LIN {X 0,Y 439.366,Z 188.757,A -85,B 0,C 180,E1 -9231.61,E2 -9231.61} C_VEL
LIN {X 0,Y 439.396,Z 188.754,A -85,B 0,C 180,E1 -9234.843,E2 -9234.843} C_VEL
LIN {X 0,Y 439.362,Z 188.757,A -85,B 0,C 180,E1 -9238.138,E2 -9238.138} C_VEL
LIN {X 0,Y 439.264,Z 188.772,A -85,B 0,C 180,E1 -9240.264,E2 -9240.264} C_VEL
LIN {X 0,Y 439.153,Z 188.786,A -85,B 0,C 180,E1 -9241.307,E2 -9241.307} C_VEL
LIN {X 0,Y 439.144,Z 192.534,A -85,B 0,C 180,E1 -9244.398,E2 -9244.398} C_VEL
LIN {X 0,Y 439.032,Z 196.208,A -85,B 0,C 180,E1 -9247.405,E2 -9247.405} C_VEL
LIN {X 0,Y 438.967,Z 200.55,A -85,B 0,C 180,E1 -9250.841,E2 -9250.841} C_VEL
LIN {X 0,Y 438.942,Z 204.965,A -85,B 0,C 180,E1 -9254.204,E2 -9254.204} C_VEL
LIN {X 0,Y 438.995,Z 210.349,A -85,B 0,C 180,E1 -9257.987,E2 -9257.987} C_VEL
LIN {X 0,Y 438.917,Z 212.924,A -85,B 0,C 180,E1 -9259.65,E2 -9259.65} C_VEL
LIN {X 0,Y 441.323,Z 223.751,A -85,B 0,C 180,E1 -9260.165,E2 -9260.165} C_VEL
LIN {X 0,Y 441.548,Z 228.336,A -85,B 0,C 180,E1 -9260.424,E2 -9260.424} C_VEL
LIN {X 0,Y 441.418,Z 237.367,A -85,B 0,C 180,E1 -9261.06,E2 -9261.06} C_VEL
LIN {X 0,Y 441.338,Z 239.701,A -85,B 0,C 180,E1 -9261.27,E2 -9261.27} C_VEL
LIN {X 0,Y 440.592,Z 243.022,A -85,B 0,C 180,E1 -9261.552,E2 -9261.552} C_VEL
LIN {X 0,Y 437.589,Z 248.036,A -85,B 0,C 180,E1 -9261.998,E2 -9261.998} C_VEL
LIN {X 0,Y 434.58,Z 252.712,A -85,B 0,C 180,E1 -9262.503,E2 -9262.503} C_VEL
LIN {X 0,Y 433.802,Z 255.354,A -85,B 0,C 180,E1 -9262.882,E2 -9262.882} C_VEL
LIN {X 0,Y 433.395,Z 261.174,A -85,B 0,C 180,E1 -9263.948,E2 -9263.948} C_VEL
LIN {X 0,Y 433.059,Z 265.059,A -85,B 0,C 180,E1 -9264.878,E2 -9264.878} C_VEL
LIN {X 0,Y 432.817,Z 269.268,A -85,B 0,C 180,E1 -9266.275,E2 -9266.275} C_VEL
LIN {X 0,Y 432.501,Z 271.224,A -85,B 0,C 180,E1 -9267.205,E2 -9267.205} C_VEL
LIN {X 0,Y 432.474,Z 272.539,A -85,B 0,C 180,E1 -9268.136,E2 -9268.136} C_VEL
LIN {X 0,Y 432.367,Z 273.322,A -85,B 0,C 180,E1 -9269.067,E2 -9269.067} C_VEL
LIN {X 0,Y 432.324,Z 273.591,A -85,B 0,C 180,E1 -9269.999,E2 -9269.999} C_VEL
LIN {X 0,Y 432.36,Z 273.368,A -85,B 0,C 180,E1 -9270.93,E2 -9270.93} C_VEL
LIN {X 0,Y 432.448,Z 272.641,A -85,B 0,C 180,E1 -9271.861,E2 -9271.861} C_VEL
LIN {X 0,Y 432.495,Z 271.382,A -85,B 0,C 180,E1 -9272.793,E2 -9272.793} C_VEL
LIN {X 0,Y 432.977,Z 268.298,A -85,B 0,C 180,E1 -9274.188,E2 -9274.188} C_VEL
LIN {X 0,Y 433.091,Z 263.642,A -85,B 0,C 180,E1 -9275.586,E2 -9275.586} C_VEL
LIN {X 0,Y 433.453,Z 260.509,A -85,B 0,C 180,E1 -9276.282,E2 -9276.282} C_VEL
LIN {X 0,Y 433.76,Z 253.871,A -85,B 0,C 180,E1 -9277.446,E2 -9277.446} C_VEL
LIN {X 0,Y 434.169,Z 246.685,A -85,B 0,C 180,E1 -9278.376,E2 -9278.376} C_VEL
LIN {X 0,Y 434.424,Z 239.235,A -85,B 0,C 180,E1 -9279.124,E2 -9279.124} C_VEL
LIN {X 0,Y 434.667,Z 230.594,A -85,B 0,C 180,E1 -9279.773,E2 -9279.773} C_VEL
LIN {X 0,Y 434.533,Z 225.553,A -85,B 0,C 180,E1 -9280.07,E2 -9280.07} C_VEL
LIN {X 0,Y 432.434,Z 216.056,A -85,B 0,C 180,E1 -9280.549,E2 -9280.549} C_VEL
LIN {X 0,Y 431.91,Z 213.531,A -85,B 0,C 180,E1 -9280.665,E2 -9280.665} C_VEL
LIN {X 0,Y 431.872,Z 209.743,A -85,B 0,C 180,E1 -9283.168,E2 -9283.168} C_VEL
LIN {X 0,Y 431.93,Z 205.419,A -85,B 0,C 180,E1 -9286.26,E2 -9286.26} C_VEL
LIN {X 0,Y 431.936,Z 201.432,A -85,B 0,C 180,E1 -9289.314,E2 -9289.314} C_VEL
LIN {X 0,Y 432.007,Z 198.074,A -85,B 0,C 180,E1 -9291.983,E2 -9291.983} C_VEL
LIN {X 0,Y 432.063,Z 194.327,A -85,B 0,C 180,E1 -9295.017,E2 -9295.017} C_VEL
LIN {X 0,Y 432.113,Z 191.814,A -85,B 0,C 180,E1 -9297.089,E2 -9297.089} C_VEL
LIN {X 0,Y 432.131,Z 190.006,A -85,B 0,C 180,E1 -9298.569,E2 -9298.569} C_VEL
LIN {X 0,Y 432.145,Z 189.659,A -85,B 0,C 180,E1 -9299.2,E2 -9299.2} C_VEL
LIN {X 0,Y 432.301,Z 189.637,A -85,B 0,C 180,E1 -9301.346,E2 -9301.346} C_VEL
LIN {X 0,Y 432.336,Z 189.63,A -85,B 0,C 180,E1 -9304.676,E2 -9304.676} C_VEL
LIN {X 0,Y 432.341,Z 189.629,A -85,B 0,C 180,E1 -9308.148,E2 -9308.148} C_VEL
LIN {X 0,Y 432.328,Z 189.632,A -85,B 0,C 180,E1 -9311.601,E2 -9311.601} C_VEL
LIN {X 0,Y 432.334,Z 189.628,A -85,B 0,C 180,E1 -9314.345,E2 -9314.345} C_VEL
LIN {X 0,Y 432.313,Z 189.635,A -85,B 0,C 180,E1 -9317.014,E2 -9317.014} C_VEL
LIN {X 0,Y 432.336,Z 189.627,A -85,B 0,C 180,E1 -9319.818,E2 -9319.818} C_VEL
LIN {X 0,Y 432.308,Z 189.634,A -85,B 0,C 180,E1 -9323.022,E2 -9323.022} C_VEL
LIN {X 0,Y 432.351,Z 189.627,A -85,B 0,C 180,E1 -9325.995,E2 -9325.995} C_VEL
LIN {X 0,Y 432.386,Z 189.622,A -85,B 0,C 180,E1 -9329.743,E2 -9329.743} C_VEL
LIN {X 0,Y 432.39,Z 189.622,A -85,B 0,C 180,E1 -9333.371,E2 -9333.371} C_VEL
LIN {X 0,Y 432.361,Z 189.626,A -85,B 0,C 180,E1 -9336.023,E2 -9336.023} C_VEL
LIN {X 0,Y 432.34,Z 189.625,A -85,B 0,C 180,E1 -9339.045,E2 -9339.045} C_VEL
LIN {X 0,Y 432.368,Z 189.629,A -85,B 0,C 180,E1 -9342.011,E2 -9342.011} C_VEL
LIN {X 0,Y 432.391,Z 189.615,A -85,B 0,C 180,E1 -9344.926,E2 -9344.926} C_VEL
LIN {X 0,Y 432.448,Z 189.617,A -85,B 0,C 180,E1 -9347.803,E2 -9347.803} C_VEL
LIN {X 0,Y 432.481,Z 189.614,A -85,B 0,C 180,E1 -9351.59,E2 -9351.59} C_VEL
LIN {X 0,Y 432.582,Z 189.594,A -85,B 0,C 180,E1 -9354.406,E2 -9354.406} C_VEL
LIN {X 0,Y 432.595,Z 189.595,A -85,B 0,C 180,E1 -9358.138,E2 -9358.138} C_VEL
LIN {X 0,Y 432.72,Z 189.573,A -85,B 0,C 180,E1 -9360,E2 -9360} C_VEL
LIN {X 0,Y 432.578,Z 189.604,A -85,B 0,C 180,E1 -9362.794,E2 -9362.794} C_VEL
LIN {X 0,Y 432.556,Z 189.604,A -85,B 0,C 180,E1 -9366.531,E2 -9366.531} C_VEL
LIN {X 0,Y 432.429,Z 189.613,A -85,B 0,C 180,E1 -9369.353,E2 -9369.353} C_VEL
LIN {X 0,Y 432.419,Z 189.616,A -85,B 0,C 180,E1 -9372.804,E2 -9372.804} C_VEL
LIN {X 0,Y 432.399,Z 189.622,A -85,B 0,C 180,E1 -9376.479,E2 -9376.479} C_VEL
LIN {X 0,Y 432.327,Z 189.637,A -85,B 0,C 180,E1 -9379.961,E2 -9379.961} C_VEL
LIN {X 0,Y 432.299,Z 189.634,A -85,B 0,C 180,E1 -9382.965,E2 -9382.965} C_VEL
LIN {X 0,Y 432.306,Z 189.638,A -85,B 0,C 180,E1 -9386.036,E2 -9386.036} C_VEL
LIN {X 0,Y 432.312,Z 189.635,A -85,B 0,C 180,E1 -9389.19,E2 -9389.19} C_VEL
LIN {X 0,Y 432.312,Z 189.632,A -85,B 0,C 180,E1 -9392.444,E2 -9392.444} C_VEL
LIN {X 0,Y 432.332,Z 189.634,A -85,B 0,C 180,E1 -9395.632,E2 -9395.632} C_VEL
LIN {X 0,Y 432.32,Z 189.636,A -85,B 0,C 180,E1 -9398.714,E2 -9398.714} C_VEL
LIN {X 0,Y 432.311,Z 189.634,A -85,B 0,C 180,E1 -9401.8,E2 -9401.8} C_VEL
LIN {X 0,Y 432.326,Z 189.632,A -85,B 0,C 180,E1 -9404.349,E2 -9404.349} C_VEL
LIN {X 0,Y 432.313,Z 189.631,A -85,B 0,C 180,E1 -9407.017,E2 -9407.017} C_VEL
LIN {X 0,Y 432.327,Z 189.634,A -85,B 0,C 180,E1 -9409.822,E2 -9409.822} C_VEL
LIN {X 0,Y 432.318,Z 189.693,A -85,B 0,C 180,E1 -9413.098,E2 -9413.098} C_VEL
LIN {X 0,Y 434.697,Z 199.485,A -85,B 0,C 180,E1 -9415.753,E2 -9415.753} C_VEL
LIN {X 0,Y 437.238,Z 210.934,A -85,B 0,C 180,E1 -9418.615,E2 -9418.615} C_VEL
LIN {X 0,Y 437.708,Z 214.124,A -85,B 0,C 180,E1 -9419.352,E2 -9419.352} C_VEL
LIN {X 0,Y 436.282,Z 228.623,A -85,B 0,C 180,E1 -9422.374,E2 -9422.374} C_VEL
LIN {X 0,Y 434.667,Z 247.312,A -85,B 0,C 180,E1 -9426.159,E2 -9426.159} C_VEL
LIN {X 0,Y 433.52,Z 264.525,A -85,B 0,C 180,E1 -9429.603,E2 -9429.603} C_VEL
LIN {X 0,Y 432.462,Z 282.864,A -85,B 0,C 180,E1 -9433.355,E2 -9433.355} C_VEL
LIN {X 0,Y 432.406,Z 284.264,A -85,B 0,C 180,E1 -9433.649,E2 -9433.649} C_VEL
LIN {X 0,Y 434.151,Z 302.397,A -85,B 0,C 180,E1 -9434.163,E2 -9434.163} C_VEL
LIN {X 0,Y 434.663,Z 314.357,A -85,B 0,C 180,E1 -9434.648,E2 -9434.648} C_VEL
LIN {X 0,Y 434.181,Z 327.38,A -85,B 0,C 180,E1 -9435.351,E2 -9435.351} C_VEL
LIN {X 0,Y 433.629,Z 339.016,A -85,B 0,C 180,E1 -9436.171,E2 -9436.171} C_VEL
LIN {X 0,Y 433.07,Z 349.53,A -85,B 0,C 180,E1 -9437.108,E2 -9437.108} C_VEL
LIN {X 0,Y 432.534,Z 360.155,A -85,B 0,C 180,E1 -9438.283,E2 -9438.283} C_VEL
LIN {X 0,Y 432.099,Z 368.825,A -85,B 0,C 180,E1 -9439.458,E2 -9439.458} C_VEL
LIN {X 0,Y 431.747,Z 377.221,A -85,B 0,C 180,E1 -9440.869,E2 -9440.869} C_VEL
LIN {X 0,Y 431.526,Z 383.96,A -85,B 0,C 180,E1 -9442.28,E2 -9442.28} C_VEL
LIN {X 0,Y 431.39,Z 389.034,A -85,B 0,C 180,E1 -9443.609,E2 -9443.609} C_VEL
LIN {X 0,Y 431.437,Z 392.806,A -85,B 0,C 180,E1 -9444.861,E2 -9444.861} C_VEL
LIN {X 0,Y 431.391,Z 395.987,A -85,B 0,C 180,E1 -9446.265,E2 -9446.265} C_VEL
LIN {X 0,Y 431.423,Z 397.549,A -85,B 0,C 180,E1 -9447.2,E2 -9447.2} C_VEL
LIN {X 0,Y 431.413,Z 398.638,A -85,B 0,C 180,E1 -9448.134,E2 -9448.134} C_VEL
LIN {X 0,Y 431.419,Z 399.29,A -85,B 0,C 180,E1 -9449.068,E2 -9449.068} C_VEL
LIN {X 0,Y 431.413,Z 399.531,A -85,B 0,C 180,E1 -9450.001,E2 -9450.001} C_VEL
LIN {X 0,Y 431.42,Z 399.348,A -85,B 0,C 180,E1 -9450.935,E2 -9450.935} C_VEL
LIN {X 0,Y 431.405,Z 398.699,A -85,B 0,C 180,E1 -9451.868,E2 -9451.868} C_VEL
LIN {X 0,Y 431.429,Z 397.639,A -85,B 0,C 180,E1 -9452.802,E2 -9452.802} C_VEL
LIN {X 0,Y 431.397,Z 396.16,A -85,B 0,C 180,E1 -9453.737,E2 -9453.737} C_VEL
LIN {X 0,Y 431.445,Z 393.062,A -85,B 0,C 180,E1 -9455.141,E2 -9455.141} C_VEL
LIN {X 0,Y 431.44,Z 388.87,A -85,B 0,C 180,E1 -9456.549,E2 -9456.549} C_VEL
LIN {X 0,Y 431.603,Z 382.413,A -85,B 0,C 180,E1 -9458.193,E2 -9458.193} C_VEL
LIN {X 0,Y 431.894,Z 375.417,A -85,B 0,C 180,E1 -9459.603,E2 -9459.603} C_VEL
LIN {X 0,Y 432.299,Z 366.74,A -85,B 0,C 180,E1 -9461.014,E2 -9461.014} C_VEL
LIN {X 0,Y 432.934,Z 355.922,A -85,B 0,C 180,E1 -9462.422,E2 -9462.422} C_VEL
LIN {X 0,Y 433.518,Z 345.135,A -85,B 0,C 180,E1 -9463.549,E2 -9463.549} C_VEL
LIN {X 0,Y 434.312,Z 333.445,A -85,B 0,C 180,E1 -9464.527,E2 -9464.527} C_VEL
LIN {X 0,Y 435.048,Z 321.115,A -85,B 0,C 180,E1 -9465.34,E2 -9465.34} C_VEL
LIN {X 0,Y 435.317,Z 311.088,A -85,B 0,C 180,E1 -9465.871,E2 -9465.871} C_VEL
LIN {X 0,Y 434.635,Z 297.333,A -85,B 0,C 180,E1 -9466.457,E2 -9466.457} C_VEL
LIN {X 0,Y 432.565,Z 280.937,A -85,B 0,C 180,E1 -9467.036,E2 -9467.036} C_VEL
LIN {X 0,Y 433.575,Z 263.253,A -85,B 0,C 180,E1 -9470.645,E2 -9470.645} C_VEL
LIN {X 0,Y 434.783,Z 246.074,A -85,B 0,C 180,E1 -9474.09,E2 -9474.09} C_VEL
LIN {X 0,Y 436.367,Z 227.495,A -85,B 0,C 180,E1 -9477.845,E2 -9477.845} C_VEL
LIN {X 0,Y 437.662,Z 214.036,A -85,B 0,C 180,E1 -9480.654,E2 -9480.654} C_VEL
LIN {X 0,Y 436.57,Z 207.954,A -85,B 0,C 180,E1 -9482.09,E2 -9482.09} C_VEL
LIN {X 0,Y 433.916,Z 196.164,A -85,B 0,C 180,E1 -9485.099,E2 -9485.099} C_VEL
LIN {X 0,Y 432.312,Z 189.638,A -85,B 0,C 180,E1 -9486.942,E2 -9486.942} C_VEL
LIN {X 0,Y 432.338,Z 189.632,A -85,B 0,C 180,E1 -9490.18,E2 -9490.18} C_VEL
LIN {X 0,Y 432.322,Z 189.634,A -85,B 0,C 180,E1 -9493.061,E2 -9493.061} C_VEL
LIN {X 0,Y 432.338,Z 189.634,A -85,B 0,C 180,E1 -9495.665,E2 -9495.665} C_VEL
LIN {X 0,Y 432.338,Z 189.633,A -85,B 0,C 180,E1 -9498.398,E2 -9498.398} C_VEL
LIN {X 0,Y 432.341,Z 189.757,A -85,B 0,C 180,E1 -9500.924,E2 -9500.924} C_VEL
LIN {X 0,Y 433.904,Z 196.549,A -85,B 0,C 180,E1 -9503.694,E2 -9503.694} C_VEL
LIN {X 0,Y 434.42,Z 199.762,A -85,B 0,C 180,E1 -9504.948,E2 -9504.948} C_VEL
LIN {X 0,Y 434.339,Z 204.343,A -85,B 0,C 180,E1 -9506.623,E2 -9506.623} C_VEL
LIN {X 0,Y 433.832,Z 213.134,A -85,B 0,C 180,E1 -9509.855,E2 -9509.855} C_VEL
LIN {X 0,Y 433.682,Z 220.548,A -85,B 0,C 180,E1 -9512.493,E2 -9512.493} C_VEL
LIN {X 0,Y 433.348,Z 229.943,A -85,B 0,C 180,E1 -9516.081,E2 -9516.081} C_VEL
LIN {X 0,Y 433.048,Z 239.208,A -85,B 0,C 180,E1 -9519.578,E2 -9519.578} C_VEL
LIN {X 0,Y 432.859,Z 246.938,A -85,B 0,C 180,E1 -9522.52,E2 -9522.52} C_VEL
LIN {X 0,Y 432.823,Z 248.27,A -85,B 0,C 180,E1 -9523.028,E2 -9523.028} C_VEL
LIN {X 0,Y 436.157,Z 261.185,A -85,B 0,C 180,E1 -9523.67,E2 -9523.67} C_VEL
LIN {X 0,Y 436.8,Z 264.746,A -85,B 0,C 180,E1 -9523.862,E2 -9523.862} C_VEL
LIN {X 0,Y 436.163,Z 278.327,A -85,B 0,C 180,E1 -9524.581,E2 -9524.581} C_VEL
LIN {X 0,Y 435.563,Z 289.849,A -85,B 0,C 180,E1 -9525.379,E2 -9525.379} C_VEL
LIN {X 0,Y 434.867,Z 300.72,A -85,B 0,C 180,E1 -9526.328,E2 -9526.328} C_VEL
LIN {X 0,Y 434.171,Z 310.523,A -85,B 0,C 180,E1 -9527.377,E2 -9527.377} C_VEL
LIN {X 0,Y 433.522,Z 319.523,A -85,B 0,C 180,E1 -9528.546,E2 -9528.546} C_VEL
LIN {X 0,Y 433.014,Z 326.938,A -85,B 0,C 180,E1 -9529.716,E2 -9529.716} C_VEL
LIN {X 0,Y 432.504,Z 334.208,A -85,B 0,C 180,E1 -9531.12,E2 -9531.12} C_VEL
LIN {X 0,Y 432.099,Z 340.07,A -85,B 0,C 180,E1 -9532.524,E2 -9532.524} C_VEL
LIN {X 0,Y 431.763,Z 344.689,A -85,B 0,C 180,E1 -9533.927,E2 -9533.927} C_VEL
LIN {X 0,Y 431.703,Z 348.178,A -85,B 0,C 180,E1 -9535.331,E2 -9535.331} C_VEL
LIN {X 0,Y 431.565,Z 349.968,A -85,B 0,C 180,E1 -9536.265,E2 -9536.265} C_VEL
LIN {X 0,Y 431.472,Z 351.286,A -85,B 0,C 180,E1 -9537.199,E2 -9537.199} C_VEL
LIN {X 0,Y 431.4,Z 352.199,A -85,B 0,C 180,E1 -9538.133,E2 -9538.133} C_VEL
LIN {X 0,Y 431.318,Z 352.722,A -85,B 0,C 180,E1 -9539.066,E2 -9539.066} C_VEL
LIN {X 0,Y 431.289,Z 352.813,A -85,B 0,C 180,E1 -9540,E2 -9540} C_VEL
LIN {X 0,Y 431.314,Z 351.753,A -85,B 0,C 180,E1 -9541.868,E2 -9541.868} C_VEL
LIN {X 0,Y 431.417,Z 350.62,A -85,B 0,C 180,E1 -9542.801,E2 -9542.801} C_VEL
LIN {X 0,Y 431.478,Z 348.099,A -85,B 0,C 180,E1 -9544.203,E2 -9544.203} C_VEL
LIN {X 0,Y 431.584,Z 344.559,A -85,B 0,C 180,E1 -9545.607,E2 -9545.607} C_VEL
LIN {X 0,Y 431.809,Z 339.391,A -85,B 0,C 180,E1 -9547.141,E2 -9547.141} C_VEL
LIN {X 0,Y 432.139,Z 332.851,A -85,B 0,C 180,E1 -9548.652,E2 -9548.652} C_VEL
LIN {X 0,Y 432.552,Z 325.23,A -85,B 0,C 180,E1 -9550.059,E2 -9550.059} C_VEL
LIN {X 0,Y 433.107,Z 315.679,A -85,B 0,C 180,E1 -9551.466,E2 -9551.466} C_VEL
LIN {X 0,Y 433.669,Z 305.897,A -85,B 0,C 180,E1 -9552.637,E2 -9552.637} C_VEL
LIN {X 0,Y 434.238,Z 294.872,A -85,B 0,C 180,E1 -9553.701,E2 -9553.701} C_VEL
LIN {X 0,Y 434.789,Z 282.839,A -85,B 0,C 180,E1 -9554.629,E2 -9554.629} C_VEL
LIN {X 0,Y 435.382,Z 269.906,A -85,B 0,C 180,E1 -9555.387,E2 -9555.387} C_VEL
LIN {X 0,Y 435.38,Z 262.377,A -85,B 0,C 180,E1 -9555.747,E2 -9555.747} C_VEL
LIN {X 0,Y 432.829,Z 248.974,A -85,B 0,C 180,E1 -9556.301,E2 -9556.301} C_VEL
LIN {X 0,Y 432.198,Z 245.514,A -85,B 0,C 180,E1 -9556.427,E2 -9556.427} C_VEL
LIN {X 0,Y 432.364,Z 236.205,A -85,B 0,C 180,E1 -9559.959,E2 -9559.959} C_VEL
LIN {X 0,Y 432.545,Z 228.361,A -85,B 0,C 180,E1 -9562.952,E2 -9562.952} C_VEL
LIN {X 0,Y 432.692,Z 220.375,A -85,B 0,C 180,E1 -9566.011,E2 -9566.011} C_VEL
LIN {X 0,Y 432.957,Z 212.189,A -85,B 0,C 180,E1 -9569.142,E2 -9569.142} C_VEL
LIN {X 0,Y 433.133,Z 203.812,A -85,B 0,C 180,E1 -9572.375,E2 -9572.375} C_VEL
LIN {X 0,Y 433.269,Z 196.593,A -85,B 0,C 180,E1 -9575.159,E2 -9575.159} C_VEL
LIN {X 0,Y 432.669,Z 191.204,A -85,B 0,C 180,E1 -9577.256,E2 -9577.256} C_VEL
LIN {X 0,Y 432.379,Z 189.628,A -85,B 0,C 180,E1 -9577.906,E2 -9577.906} C_VEL
LIN {X 0,Y 432.326,Z 189.633,A -85,B 0,C 180,E1 -9580.561,E2 -9580.561} C_VEL
LIN {X 0,Y 432.319,Z 189.634,A -85,B 0,C 180,E1 -9583.061,E2 -9583.061} C_VEL
LIN {X 0,Y 432.338,Z 189.631,A -85,B 0,C 180,E1 -9585.664,E2 -9585.664} C_VEL
LIN {X 0,Y 432.338,Z 189.631,A -85,B 0,C 180,E1 -9588.398,E2 -9588.398} C_VEL
LIN {X 0,Y 432.33,Z 189.634,A -85,B 0,C 180,E1 -9591.848,E2 -9591.848} C_VEL
LIN {X 0,Y 432.33,Z 189.636,A -85,B 0,C 180,E1 -9595.321,E2 -9595.321} C_VEL
LIN {X 0,Y 432.3,Z 189.639,A -85,B 0,C 180,E1 -9598.651,E2 -9598.651} C_VEL
LIN {X 0,Y 432.125,Z 189.881,A -85,B 0,C 180,E1 -9601.432,E2 -9601.432} C_VEL
LIN {X 0,Y 432.115,Z 192.93,A -85,B 0,C 180,E1 -9603.95,E2 -9603.95} C_VEL
LIN {X 0,Y 432.005,Z 196.684,A -85,B 0,C 180,E1 -9607.017,E2 -9607.017} C_VEL
LIN {X 0,Y 431.941,Z 201.27,A -85,B 0,C 180,E1 -9610.684,E2 -9610.684} C_VEL
LIN {X 0,Y 431.898,Z 205.538,A -85,B 0,C 180,E1 -9613.94,E2 -9613.94} C_VEL
LIN {X 0,Y 431.944,Z 211,A -85,B 0,C 180,E1 -9617.788,E2 -9617.788} C_VEL
LIN {X 0,Y 431.898,Z 213.618,A -85,B 0,C 180,E1 -9619.451,E2 -9619.451} C_VEL
LIN {X 0,Y 434.257,Z 224.071,A -85,B 0,C 180,E1 -9619.939,E2 -9619.939} C_VEL
LIN {X 0,Y 434.685,Z 227.626,A -85,B 0,C 180,E1 -9620.143,E2 -9620.143} C_VEL
LIN {X 0,Y 434.506,Z 236.893,A -85,B 0,C 180,E1 -9620.774,E2 -9620.774} C_VEL
LIN {X 0,Y 434.227,Z 244.517,A -85,B 0,C 180,E1 -9621.472,E2 -9621.472} C_VEL
LIN {X 0,Y 433.86,Z 251.526,A -85,B 0,C 180,E1 -9622.319,E2 -9622.319} C_VEL
LIN {X 0,Y 433.802,Z 255.354,A -85,B 0,C 180,E1 -9622.882,E2 -9622.882} C_VEL
LIN {X 0,Y 433.001,Z 257.885,A -85,B 0,C 180,E1 -9623.282,E2 -9623.282} C_VEL
LIN {X 0,Y 429.88,Z 261.704,A -85,B 0,C 180,E1 -9623.901,E2 -9623.901} C_VEL
LIN {X 0,Y 426.797,Z 265.096,A -85,B 0,C 180,E1 -9624.567,E2 -9624.567} C_VEL
LIN {X 0,Y 426.058,Z 266.865,A -85,B 0,C 180,E1 -9625.034,E2 -9625.034} C_VEL
LIN {X 0,Y 425.815,Z 270.255,A -85,B 0,C 180,E1 -9626.213,E2 -9626.213} C_VEL
LIN {X 0,Y 425.487,Z 272.204,A -85,B 0,C 180,E1 -9627.158,E2 -9627.158} C_VEL
LIN {X 0,Y 425.456,Z 273.515,A -85,B 0,C 180,E1 -9628.106,E2 -9628.106} C_VEL
LIN {X 0,Y 425.345,Z 274.296,A -85,B 0,C 180,E1 -9629.052,E2 -9629.052} C_VEL
LIN {X 0,Y 425.3,Z 274.565,A -85,B 0,C 180,E1 -9629.999,E2 -9629.999} C_VEL
LIN {X 0,Y 425.339,Z 274.342,A -85,B 0,C 180,E1 -9630.946,E2 -9630.946} C_VEL
LIN {X 0,Y 425.432,Z 273.616,A -85,B 0,C 180,E1 -9631.892,E2 -9631.892} C_VEL
LIN {X 0,Y 425.482,Z 272.362,A -85,B 0,C 180,E1 -9632.839,E2 -9632.839} C_VEL
LIN {X 0,Y 425.981,Z 269.288,A -85,B 0,C 180,E1 -9634.256,E2 -9634.256} C_VEL
LIN {X 0,Y 426.098,Z 264.654,A -85,B 0,C 180,E1 -9635.678,E2 -9635.678} C_VEL
LIN {X 0,Y 426.473,Z 261.542,A -85,B 0,C 180,E1 -9636.385,E2 -9636.385} C_VEL
LIN {X 0,Y 426.807,Z 254.956,A -85,B 0,C 180,E1 -9637.568,E2 -9637.568} C_VEL
LIN {X 0,Y 427.234,Z 247.821,A -85,B 0,C 180,E1 -9638.513,E2 -9638.513} C_VEL
LIN {X 0,Y 427.507,Z 240.315,A -85,B 0,C 180,E1 -9639.284,E2 -9639.284} C_VEL
LIN {X 0,Y 427.786,Z 231.984,A -85,B 0,C 180,E1 -9639.932,E2 -9639.932} C_VEL
LIN {X 0,Y 427.696,Z 227.044,A -85,B 0,C 180,E1 -9640.233,E2 -9640.233} C_VEL
LIN {X 0,Y 425.517,Z 216.936,A -85,B 0,C 180,E1 -9640.76,E2 -9640.76} C_VEL
LIN {X 0,Y 424.854,Z 214.126,A -85,B 0,C 180,E1 -9640.905,E2 -9640.905} C_VEL
LIN {X 0,Y 424.827,Z 210.378,A -85,B 0,C 180,E1 -9643.39,E2 -9643.39} C_VEL
LIN {X 0,Y 424.894,Z 206.183,A -85,B 0,C 180,E1 -9646.391,E2 -9646.391} C_VEL
LIN {X 0,Y 424.887,Z 202.17,A -85,B 0,C 180,E1 -9649.467,E2 -9649.467} C_VEL
LIN {X 0,Y 424.95,Z 198.543,A -85,B 0,C 180,E1 -9652.356,E2 -9652.356} C_VEL
LIN {X 0,Y 425.048,Z 194.746,A -85,B 0,C 180,E1 -9655.46,E2 -9655.46} C_VEL
LIN {X 0,Y 425.101,Z 190.885,A -85,B 0,C 180,E1 -9658.647,E2 -9658.647} C_VEL
LIN {X 0,Y 425.239,Z 190.515,A -85,B 0,C 180,E1 -9660.818,E2 -9660.818} C_VEL
LIN {X 0,Y 425.308,Z 190.506,A -85,B 0,C 180,E1 -9664.287,E2 -9664.287} C_VEL
LIN {X 0,Y 425.281,Z 190.511,A -85,B 0,C 180,E1 -9667.692,E2 -9667.692} C_VEL
LIN {X 0,Y 425.276,Z 190.509,A -85,B 0,C 180,E1 -9670.519,E2 -9670.519} C_VEL
LIN {X 0,Y 425.257,Z 190.513,A -85,B 0,C 180,E1 -9673.35,E2 -9673.35} C_VEL
LIN {X 0,Y 425.25,Z 190.513,A -85,B 0,C 180,E1 -9676.648,E2 -9676.648} C_VEL
LIN {X 0,Y 425.289,Z 190.505,A -85,B 0,C 180,E1 -9679.873,E2 -9679.873} C_VEL
LIN {X 0,Y 425.277,Z 190.51,A -85,B 0,C 180,E1 -9682.486,E2 -9682.486} C_VEL
LIN {X 0,Y 425.299,Z 190.504,A -85,B 0,C 180,E1 -9685.816,E2 -9685.816} C_VEL
LIN {X 0,Y 425.295,Z 190.505,A -85,B 0,C 180,E1 -9689.235,E2 -9689.235} C_VEL
LIN {X 0,Y 425.341,Z 190.504,A -85,B 0,C 180,E1 -9692.442,E2 -9692.442} C_VEL
LIN {X 0,Y 425.341,Z 190.496,A -85,B 0,C 180,E1 -9695.601,E2 -9695.601} C_VEL
LIN {X 0,Y 425.283,Z 190.504,A -85,B 0,C 180,E1 -9698.681,E2 -9698.681} C_VEL
LIN {X 0,Y 425.323,Z 190.506,A -85,B 0,C 180,E1 -9701.702,E2 -9701.702} C_VEL
LIN {X 0,Y 425.345,Z 190.492,A -85,B 0,C 180,E1 -9704.67,E2 -9704.67} C_VEL
LIN {X 0,Y 425.401,Z 190.497,A -85,B 0,C 180,E1 -9707.598,E2 -9707.598} C_VEL
LIN {X 0,Y 425.431,Z 190.491,A -85,B 0,C 180,E1 -9711.45,E2 -9711.45} C_VEL
LIN {X 0,Y 425.538,Z 190.471,A -85,B 0,C 180,E1 -9714.313,E2 -9714.313} C_VEL
LIN {X 0,Y 425.564,Z 190.471,A -85,B 0,C 180,E1 -9718.107,E2 -9718.107} C_VEL
LIN {X 0,Y 425.69,Z 190.449,A -85,B 0,C 180,E1 -9720,E2 -9720} C_VEL
LIN {X 0,Y 425.531,Z 190.481,A -85,B 0,C 180,E1 -9722.84,E2 -9722.84} C_VEL
LIN {X 0,Y 425.515,Z 190.483,A -85,B 0,C 180,E1 -9726.639,E2 -9726.639} C_VEL
LIN {X 0,Y 425.387,Z 190.489,A -85,B 0,C 180,E1 -9729.51,E2 -9729.51} C_VEL
LIN {X 0,Y 425.381,Z 190.492,A -85,B 0,C 180,E1 -9732.904,E2 -9732.904} C_VEL
LIN {X 0,Y 425.349,Z 190.499,A -85,B 0,C 180,E1 -9736.605,E2 -9736.605} C_VEL
LIN {X 0,Y 425.316,Z 190.506,A -85,B 0,C 180,E1 -9739.636,E2 -9739.636} C_VEL
LIN {X 0,Y 425.275,Z 190.512,A -85,B 0,C 180,E1 -9742.339,E2 -9742.339} C_VEL
LIN {X 0,Y 425.248,Z 190.516,A -85,B 0,C 180,E1 -9745.448,E2 -9745.448} C_VEL
LIN {X 0,Y 425.289,Z 190.508,A -85,B 0,C 180,E1 -9748.859,E2 -9748.859} C_VEL
LIN {X 0,Y 425.254,Z 190.513,A -85,B 0,C 180,E1 -9751.928,E2 -9751.928} C_VEL
LIN {X 0,Y 425.287,Z 190.51,A -85,B 0,C 180,E1 -9755.337,E2 -9755.337} C_VEL
LIN {X 0,Y 425.274,Z 190.516,A -85,B 0,C 180,E1 -9758.901,E2 -9758.901} C_VEL
LIN {X 0,Y 425.271,Z 190.511,A -85,B 0,C 180,E1 -9761.958,E2 -9761.958} C_VEL
LIN {X 0,Y 425.277,Z 190.51,A -85,B 0,C 180,E1 -9765.284,E2 -9765.284} C_VEL
LIN {X 0,Y 425.267,Z 190.507,A -85,B 0,C 180,E1 -9768.623,E2 -9768.623} C_VEL
LIN {X 0,Y 425.3,Z 190.503,A -85,B 0,C 180,E1 -9771.104,E2 -9771.104} C_VEL
LIN {X 0,Y 425.309,Z 190.713,A -85,B 0,C 180,E1 -9772.684,E2 -9772.684} C_VEL
LIN {X 0,Y 427.903,Z 201.469,A -85,B 0,C 180,E1 -9775.679,E2 -9775.679} C_VEL
LIN {X 0,Y 430.377,Z 212.6,A -85,B 0,C 180,E1 -9778.498,E2 -9778.498} C_VEL
LIN {X 0,Y 430.803,Z 216.222,A -85,B 0,C 180,E1 -9779.351,E2 -9779.351} C_VEL
LIN {X 0,Y 429.104,Z 232.027,A -85,B 0,C 180,E1 -9782.705,E2 -9782.705} C_VEL
LIN {X 0,Y 427.623,Z 249.211,A -85,B 0,C 180,E1 -9786.257,E2 -9786.257} C_VEL
LIN {X 0,Y 426.408,Z 266.239,A -85,B 0,C 180,E1 -9789.751,E2 -9789.751} C_VEL
LIN {X 0,Y 425.359,Z 283.693,A -85,B 0,C 180,E1 -9793.418,E2 -9793.418} C_VEL
LIN {X 0,Y 427.186,Z 302.416,A -85,B 0,C 180,E1 -9793.96,E2 -9793.96} C_VEL
LIN {X 0,Y 427.699,Z 315.433,A -85,B 0,C 180,E1 -9794.514,E2 -9794.514} C_VEL
LIN {X 0,Y 427.147,Z 328.088,A -85,B 0,C 180,E1 -9795.226,E2 -9795.226} C_VEL
LIN {X 0,Y 426.604,Z 339.456,A -85,B 0,C 180,E1 -9796.06,E2 -9796.06} C_VEL
LIN {X 0,Y 426.03,Z 349.777,A -85,B 0,C 180,E1 -9797.01,E2 -9797.01} C_VEL
LIN {X 0,Y 425.505,Z 359.342,A -85,B 0,C 180,E1 -9798.086,E2 -9798.086} C_VEL
LIN {X 0,Y 425.05,Z 368.084,A -85,B 0,C 180,E1 -9799.281,E2 -9799.281} C_VEL
LIN {X 0,Y 424.693,Z 376.568,A -85,B 0,C 180,E1 -9800.716,E2 -9800.716} C_VEL
LIN {X 0,Y 424.438,Z 383.356,A -85,B 0,C 180,E1 -9802.15,E2 -9802.15} C_VEL
LIN {X 0,Y 424.292,Z 388.951,A -85,B 0,C 180,E1 -9803.641,E2 -9803.641} C_VEL
LIN {X 0,Y 424.32,Z 393.495,A -85,B 0,C 180,E1 -9805.251,E2 -9805.251} C_VEL
LIN {X 0,Y 424.296,Z 395.505,A -85,B 0,C 180,E1 -9806.202,E2 -9806.202} C_VEL
LIN {X 0,Y 424.349,Z 397.084,A -85,B 0,C 180,E1 -9807.153,E2 -9807.153} C_VEL
LIN {X 0,Y 424.328,Z 398.205,A -85,B 0,C 180,E1 -9808.103,E2 -9808.103} C_VEL
LIN {X 0,Y 424.354,Z 398.871,A -85,B 0,C 180,E1 -9809.052,E2 -9809.052} C_VEL
LIN {X 0,Y 424.347,Z 399.125,A -85,B 0,C 180,E1 -9810.001,E2 -9810.001} C_VEL
LIN {X 0,Y 424.355,Z 398.964,A -85,B 0,C 180,E1 -9810.95,E2 -9810.95} C_VEL
LIN {X 0,Y 424.32,Z 398.334,A -85,B 0,C 180,E1 -9811.9,E2 -9811.9} C_VEL
LIN {X 0,Y 424.354,Z 397.284,A -85,B 0,C 180,E1 -9812.849,E2 -9812.849} C_VEL
LIN {X 0,Y 424.297,Z 395.814,A -85,B 0,C 180,E1 -9813.8,E2 -9813.8} C_VEL
LIN {X 0,Y 424.346,Z 392.74,A -85,B 0,C 180,E1 -9815.228,E2 -9815.228} C_VEL
LIN {X 0,Y 424.355,Z 388.581,A -85,B 0,C 180,E1 -9816.659,E2 -9816.659} C_VEL
LIN {X 0,Y 424.532,Z 382.177,A -85,B 0,C 180,E1 -9818.33,E2 -9818.33} C_VEL
LIN {X 0,Y 424.848,Z 375.221,A -85,B 0,C 180,E1 -9819.763,E2 -9819.763} C_VEL
LIN {X 0,Y 425.313,Z 366.639,A -85,B 0,C 180,E1 -9821.197,E2 -9821.197} C_VEL
LIN {X 0,Y 425.981,Z 356.054,A -85,B 0,C 180,E1 -9822.609,E2 -9822.609} C_VEL
LIN {X 0,Y 426.529,Z 346.407,A -85,B 0,C 180,E1 -9823.666,E2 -9823.666} C_VEL
LIN {X 0,Y 427.365,Z 335.307,A -85,B 0,C 180,E1 -9824.647,E2 -9824.647} C_VEL
LIN {X 0,Y 428.153,Z 323.684,A -85,B 0,C 180,E1 -9825.471,E2 -9825.471} C_VEL
LIN {X 0,Y 428.588,Z 312.182,A -85,B 0,C 180,E1 -9826.127,E2 -9826.127} C_VEL
LIN {X 0,Y 427.953,Z 298.246,A -85,B 0,C 180,E1 -9826.761,E2 -9826.761} C_VEL
LIN {X 0,Y 425.602,Z 279.414,A -85,B 0,C 180,E1 -9827.479,E2 -9827.479} C_VEL
LIN {X 0,Y 426.742,Z 261.382,A -85,B 0,C 180,E1 -9831.244,E2 -9831.244} C_VEL
LIN {X 0,Y 428.247,Z 241.821,A -85,B 0,C 180,E1 -9835.259,E2 -9835.259} C_VEL
LIN {X 0,Y 429.854,Z 224.627,A -85,B 0,C 180,E1 -9838.838,E2 -9838.838} C_VEL
LIN {X 0,Y 430.774,Z 216.131,A -85,B 0,C 180,E1 -9840.654,E2 -9840.654} C_VEL
LIN {X 0,Y 430.066,Z 211.245,A -85,B 0,C 180,E1 -9841.813,E2 -9841.813} C_VEL
LIN {X 0,Y 427.173,Z 198.288,A -85,B 0,C 180,E1 -9845.159,E2 -9845.159} C_VEL
LIN {X 0,Y 425.289,Z 190.513,A -85,B 0,C 180,E1 -9847.396,E2 -9847.396} C_VEL
LIN {X 0,Y 425.285,Z 190.513,A -85,B 0,C 180,E1 -9850.521,E2 -9850.521} C_VEL
LIN {X 0,Y 425.263,Z 190.515,A -85,B 0,C 180,E1 -9853.351,E2 -9853.351} C_VEL
LIN {X 0,Y 425.262,Z 190.514,A -85,B 0,C 180,E1 -9856.65,E2 -9856.65} C_VEL
LIN {X 0,Y 425.298,Z 190.513,A -85,B 0,C 180,E1 -9859.983,E2 -9859.983} C_VEL
LIN {X 0,Y 426.974,Z 197.559,A -85,B 0,C 180,E1 -9863.073,E2 -9863.073} C_VEL
LIN {X 0,Y 427.709,Z 202.04,A -85,B 0,C 180,E1 -9864.893,E2 -9864.893} C_VEL
LIN {X 0,Y 427.471,Z 208.041,A -85,B 0,C 180,E1 -9867.143,E2 -9867.143} C_VEL
LIN {X 0,Y 426.919,Z 217.582,A -85,B 0,C 180,E1 -9870.751,E2 -9870.751} C_VEL
LIN {X 0,Y 426.697,Z 225.3,A -85,B 0,C 180,E1 -9873.595,E2 -9873.595} C_VEL
LIN {X 0,Y 426.393,Z 233.328,A -85,B 0,C 180,E1 -9876.698,E2 -9876.698} C_VEL
LIN {X 0,Y 426.088,Z 242.155,A -85,B 0,C 180,E1 -9880.082,E2 -9880.082} C_VEL
LIN {X 0,Y 425.922,Z 248.884,A -85,B 0,C 180,E1 -9882.644,E2 -9882.644} C_VEL
LIN {X 0,Y 429.274,Z 261.187,A -85,B 0,C 180,E1 -9883.29,E2 -9883.29} C_VEL
LIN {X 0,Y 430.116,Z 267.448,A -85,B 0,C 180,E1 -9883.636,E2 -9883.636} C_VEL
LIN {X 0,Y 429.457,Z 279.954,A -85,B 0,C 180,E1 -9884.335,E2 -9884.335} C_VEL
LIN {X 0,Y 428.692,Z 292.44,A -85,B 0,C 180,E1 -9885.251,E2 -9885.251} C_VEL
LIN {X 0,Y 427.897,Z 304.151,A -85,B 0,C 180,E1 -9886.343,E2 -9886.343} C_VEL
LIN {X 0,Y 426.939,Z 315.244,A -85,B 0,C 180,E1 -9887.643,E2 -9887.643} C_VEL
LIN {X 0,Y 426.359,Z 323.451,A -85,B 0,C 180,E1 -9888.832,E2 -9888.832} C_VEL
LIN {X 0,Y 425.848,Z 331.469,A -85,B 0,C 180,E1 -9890.261,E2 -9890.261} C_VEL
LIN {X 0,Y 425.352,Z 336.991,A -85,B 0,C 180,E1 -9891.448,E2 -9891.448} C_VEL
LIN {X 0,Y 425.016,Z 342.171,A -85,B 0,C 180,E1 -9892.822,E2 -9892.822} C_VEL
LIN {X 0,Y 424.571,Z 346.536,A -85,B 0,C 180,E1 -9894.3,E2 -9894.3} C_VEL
LIN {X 0,Y 424.657,Z 348.713,A -85,B 0,C 180,E1 -9895.253,E2 -9895.253} C_VEL
LIN {X 0,Y 424.513,Z 350.473,A -85,B 0,C 180,E1 -9896.203,E2 -9896.203} C_VEL
LIN {X 0,Y 424.402,Z 351.763,A -85,B 0,C 180,E1 -9897.152,E2 -9897.152} C_VEL
LIN {X 0,Y 424.318,Z 352.655,A -85,B 0,C 180,E1 -9898.102,E2 -9898.102} C_VEL
LIN {X 0,Y 424.245,Z 353.153,A -85,B 0,C 180,E1 -9899.051,E2 -9899.051} C_VEL
LIN {X 0,Y 424.2,Z 353.207,A -85,B 0,C 180,E1 -9900,E2 -9900} C_VEL
LIN {X 0,Y 424.237,Z 352.1,A -85,B 0,C 180,E1 -9901.899,E2 -9901.899} C_VEL
LIN {X 0,Y 424.35,Z 350.929,A -85,B 0,C 180,E1 -9902.848,E2 -9902.848} C_VEL
LIN {X 0,Y 424.387,Z 348.361,A -85,B 0,C 180,E1 -9904.274,E2 -9904.274} C_VEL
LIN {X 0,Y 424.519,Z 344.762,A -85,B 0,C 180,E1 -9905.701,E2 -9905.701} C_VEL
LIN {X 0,Y 424.754,Z 339.211,A -85,B 0,C 180,E1 -9907.344,E2 -9907.344} C_VEL
LIN {X 0,Y 425.107,Z 332.924,A -85,B 0,C 180,E1 -9908.796,E2 -9908.796} C_VEL
LIN {X 0,Y 425.532,Z 325.2,A -85,B 0,C 180,E1 -9910.227,E2 -9910.227} C_VEL
LIN {X 0,Y 426.13,Z 315.567,A -85,B 0,C 180,E1 -9911.656,E2 -9911.656} C_VEL
LIN {X 0,Y 426.729,Z 305.652,A -85,B 0,C 180,E1 -9912.846,E2 -9912.846} C_VEL
LIN {X 0,Y 427.329,Z 293.819,A -85,B 0,C 180,E1 -9913.988,E2 -9913.988} C_VEL
LIN {X 0,Y 427.91,Z 282.265,A -85,B 0,C 180,E1 -9914.87,E2 -9914.87} C_VEL
LIN {X 0,Y 428.511,Z 269.117,A -85,B 0,C 180,E1 -9915.64,E2 -9915.64} C_VEL
LIN {X 0,Y 428.553,Z 264.079,A -85,B 0,C 180,E1 -9915.883,E2 -9915.883} C_VEL
LIN {X 0,Y 426.129,Z 251.066,A -85,B 0,C 180,E1 -9916.456,E2 -9916.456} C_VEL
LIN {X 0,Y 425.192,Z 245.834,A -85,B 0,C 180,E1 -9916.642,E2 -9916.642} C_VEL
LIN {X 0,Y 425.338,Z 236.254,A -85,B 0,C 180,E1 -9920.303,E2 -9920.303} C_VEL
LIN {X 0,Y 425.533,Z 228.316,A -85,B 0,C 180,E1 -9923.352,E2 -9923.352} C_VEL
LIN {X 0,Y 425.794,Z 218.947,A -85,B 0,C 180,E1 -9926.961,E2 -9926.961} C_VEL
LIN {X 0,Y 426.012,Z 210.545,A -85,B 0,C 180,E1 -9930.21,E2 -9930.21} C_VEL
LIN {X 0,Y 426.21,Z 201.994,A -85,B 0,C 180,E1 -9933.532,E2 -9933.532} C_VEL
LIN {X 0,Y 426.119,Z 195.407,A -85,B 0,C 180,E1 -9936.082,E2 -9936.082} C_VEL
LIN {X 0,Y 425.344,Z 190.505,A -85,B 0,C 180,E1 -9938.063,E2 -9938.063} C_VEL
LIN {X 0,Y 425.273,Z 190.513,A -85,B 0,C 180,E1 -9941.379,E2 -9941.379} C_VEL
LIN {X 0,Y 425.29,Z 190.507,A -85,B 0,C 180,E1 -9944.716,E2 -9944.716} C_VEL
LIN {X 0,Y 425.295,Z 190.509,A -85,B 0,C 180,E1 -9948.041,E2 -9948.041} C_VEL
LIN {X 0,Y 425.293,Z 190.511,A -85,B 0,C 180,E1 -9951.1,E2 -9951.1} C_VEL
LIN {X 0,Y 425.297,Z 190.51,A -85,B 0,C 180,E1 -9954.663,E2 -9954.663} C_VEL
LIN {X 0,Y 425.255,Z 190.514,A -85,B 0,C 180,E1 -9958.071,E2 -9958.071} C_VEL
LIN {X 0,Y 425.176,Z 190.527,A -85,B 0,C 180,E1 -9960.271,E2 -9960.271} C_VEL
LIN {X 0,Y 425.097,Z 190.755,A -85,B 0,C 180,E1 -9961.35,E2 -9961.35} C_VEL
LIN {X 0,Y 425.055,Z 194.605,A -85,B 0,C 180,E1 -9964.538,E2 -9964.538} C_VEL
LIN {X 0,Y 424.959,Z 198.622,A -85,B 0,C 180,E1 -9967.84,E2 -9967.84} C_VEL
LIN {X 0,Y 424.917,Z 202.219,A -85,B 0,C 180,E1 -9970.682,E2 -9970.682} C_VEL
LIN {X 0,Y 424.862,Z 206.115,A -85,B 0,C 180,E1 -9973.666,E2 -9973.666} C_VEL
LIN {X 0,Y 424.908,Z 211.653,A -85,B 0,C 180,E1 -9977.582,E2 -9977.582} C_VEL
LIN {X 0,Y 424.891,Z 214.322,A -85,B 0,C 180,E1 -9979.229,E2 -9979.229} C_VEL
LIN {X 0,Y 427.184,Z 224.363,A -85,B 0,C 180,E1 -9979.704,E2 -9979.704} C_VEL
LIN {X 0,Y 427.77,Z 229.089,A -85,B 0,C 180,E1 -9979.982,E2 -9979.982} C_VEL
LIN {X 0,Y 427.602,Z 238.944,A -85,B 0,C 180,E1 -9980.688,E2 -9980.688} C_VEL
LIN {X 0,Y 427.259,Z 246.979,A -85,B 0,C 180,E1 -9981.485,E2 -9981.485} C_VEL
LIN {X 0,Y 426.914,Z 252.618,A -85,B 0,C 180,E1 -9982.193,E2 -9982.193} C_VEL
LIN {X 0,Y 426.793,Z 257.256,A -85,B 0,C 180,E1 -9982.905,E2 -9982.905} C_VEL
LIN {X 0,Y 426.415,Z 262.205,A -85,B 0,C 180,E1 -9983.849,E2 -9983.849} C_VEL
LIN {X 0,Y 426.065,Z 266.066,A -85,B 0,C 180,E1 -9984.794,E2 -9984.794} C_VEL
LIN {X 0,Y 426.058,Z 266.865,A -85,B 0,C 180,E1 -9985.034,E2 -9985.034} C_VEL
LIN {X 0,Y 425.327,Z 268.506,A -85,B 0,C 180,E1 -9985.513,E2 -9985.513} C_VEL
LIN {X 0,Y 422.27,Z 270.928,A -85,B 0,C 180,E1 -9986.26,E2 -9986.26} C_VEL
LIN {X 0,Y 419.191,Z 272.957,A -85,B 0,C 180,E1 -9987.036,E2 -9987.036} C_VEL
LIN {X 0,Y 418.442,Z 273.792,A -85,B 0,C 180,E1 -9987.558,E2 -9987.558} C_VEL
LIN {X 0,Y 418.323,Z 275.271,A -85,B 0,C 180,E1 -9989.036,E2 -9989.036} C_VEL
LIN {X 0,Y 418.276,Z 275.539,A -85,B 0,C 180,E1 -9989.999,E2 -9989.999} C_VEL
LIN {X 0,Y 418.316,Z 275.315,A -85,B 0,C 180,E1 -9990.961,E2 -9990.961} C_VEL
LIN {X 0,Y 418.416,Z 274.591,A -85,B 0,C 180,E1 -9991.924,E2 -9991.924} C_VEL
LIN {X 0,Y 418.468,Z 273.341,A -85,B 0,C 180,E1 -9992.887,E2 -9992.887} C_VEL
LIN {X 0,Y 418.985,Z 270.277,A -85,B 0,C 180,E1 -9994.328,E2 -9994.328} C_VEL
LIN {X 0,Y 419.106,Z 265.664,A -85,B 0,C 180,E1 -9995.773,E2 -9995.773} C_VEL
LIN {X 0,Y 419.495,Z 262.571,A -85,B 0,C 180,E1 -9996.492,E2 -9996.492} C_VEL
LIN {X 0,Y 419.856,Z 256.034,A -85,B 0,C 180,E1 -9997.694,E2 -9997.694} C_VEL
LIN {X 0,Y 420.311,Z 248.951,A -85,B 0,C 180,E1 -9998.654,E2 -9998.654} C_VEL
LIN {X 0,Y 420.592,Z 241.418,A -85,B 0,C 180,E1 -9999.448,E2 -9999.448} C_VEL
LIN {X 0,Y 420.89,Z 234,A -85,B 0,C 180,E1 -10000.048,E2 -10000.048} C_VEL
LIN {X 0,Y 420.743,Z 227.679,A -85,B 0,C 180,E1 -10000.453,E2 -10000.453} C_VEL
LIN {X 0,Y 418.535,Z 217.729,A -85,B 0,C 180,E1 -10000.983,E2 -10000.983} C_VEL
LIN {X 0,Y 417.848,Z 214.766,A -85,B 0,C 180,E1 -10001.121,E2 -10001.121} C_VEL
LIN {X 0,Y 417.793,Z 211.019,A -85,B 0,C 180,E1 -10003.62,E2 -10003.62} C_VEL
LIN {X 0,Y 417.845,Z 206.845,A -85,B 0,C 180,E1 -10006.613,E2 -10006.613} C_VEL
LIN {X 0,Y 417.863,Z 202.889,A -85,B 0,C 180,E1 -10009.655,E2 -10009.655} C_VEL
LIN {X 0,Y 417.911,Z 199.026,A -85,B 0,C 180,E1 -10012.753,E2 -10012.753} C_VEL
LIN {X 0,Y 418.022,Z 195.186,A -85,B 0,C 180,E1 -10015.919,E2 -10015.919} C_VEL
LIN {X 0,Y 418.072,Z 191.411,A -85,B 0,C 180,E1 -10019.175,E2 -10019.175} C_VEL
LIN {X 0,Y 418.183,Z 191.396,A -85,B 0,C 180,E1 -10021.397,E2 -10021.397} C_VEL
LIN {X 0,Y 418.261,Z 191.384,A -85,B 0,C 180,E1 -10024.579,E2 -10024.579} C_VEL
LIN {X 0,Y 418.229,Z 191.389,A -85,B 0,C 180,E1 -10027.833,E2 -10027.833} C_VEL
LIN {X 0,Y 418.217,Z 191.392,A -85,B 0,C 180,E1 -10030.946,E2 -10030.946} C_VEL
LIN {X 0,Y 418.21,Z 191.388,A -85,B 0,C 180,E1 -10033.729,E2 -10033.729} C_VEL
LIN {X 0,Y 418.202,Z 191.391,A -85,B 0,C 180,E1 -10036.447,E2 -10036.447} C_VEL
LIN {X 0,Y 418.218,Z 191.388,A -85,B 0,C 180,E1 -10039.129,E2 -10039.129} C_VEL
LIN {X 0,Y 418.228,Z 191.387,A -85,B 0,C 180,E1 -10042.164,E2 -10042.164} C_VEL
LIN {X 0,Y 418.257,Z 191.381,A -85,B 0,C 180,E1 -10045.419,E2 -10045.419} C_VEL
LIN {X 0,Y 418.214,Z 191.391,A -85,B 0,C 180,E1 -10048.604,E2 -10048.604} C_VEL
LIN {X 0,Y 418.286,Z 191.38,A -85,B 0,C 180,E1 -10051.936,E2 -10051.936} C_VEL
LIN {X 0,Y 418.279,Z 191.373,A -85,B 0,C 180,E1 -10055.162,E2 -10055.162} C_VEL
LIN {X 0,Y 418.224,Z 191.386,A -85,B 0,C 180,E1 -10058.303,E2 -10058.303} C_VEL
LIN {X 0,Y 418.273,Z 191.38,A -85,B 0,C 180,E1 -10061.383,E2 -10061.383} C_VEL
LIN {X 0,Y 418.299,Z 191.37,A -85,B 0,C 180,E1 -10064.406,E2 -10064.406} C_VEL
LIN {X 0,Y 418.344,Z 191.376,A -85,B 0,C 180,E1 -10067.385,E2 -10067.385} C_VEL
LIN {X 0,Y 418.331,Z 191.366,A -85,B 0,C 180,E1 -10070.328,E2 -10070.328} C_VEL
LIN {X 0,Y 418.475,Z 191.359,A -85,B 0,C 180,E1 -10073.249,E2 -10073.249} C_VEL
LIN {X 0,Y 418.327,Z 191.371,A -85,B 0,C 180,E1 -10075.181,E2 -10075.181} C_VEL
LIN {X 0,Y 418.533,Z 191.347,A -85,B 0,C 180,E1 -10078.075,E2 -10078.075} C_VEL
LIN {X 0,Y 418.66,Z 191.324,A -85,B 0,C 180,E1 -10080,E2 -10080} C_VEL
LIN {X 0,Y 418.486,Z 191.358,A -85,B 0,C 180,E1 -10082.888,E2 -10082.888} C_VEL
LIN {X 0,Y 418.478,Z 191.361,A -85,B 0,C 180,E1 -10086.751,E2 -10086.751} C_VEL
LIN {X 0,Y 418.388,Z 191.365,A -85,B 0,C 180,E1 -10088.695,E2 -10088.695} C_VEL
LIN {X 0,Y 418.343,Z 191.371,A -85,B 0,C 180,E1 -10092.615,E2 -10092.615} C_VEL
LIN {X 0,Y 418.289,Z 191.38,A -85,B 0,C 180,E1 -10095.595,E2 -10095.595} C_VEL
LIN {X 0,Y 418.263,Z 191.384,A -85,B 0,C 180,E1 -10098.618,E2 -10098.618} C_VEL
LIN {X 0,Y 418.222,Z 191.392,A -85,B 0,C 180,E1 -10101.697,E2 -10101.697} C_VEL
LIN {X 0,Y 418.232,Z 191.387,A -85,B 0,C 180,E1 -10104.853,E2 -10104.853} C_VEL
LIN {X 0,Y 418.196,Z 191.394,A -85,B 0,C 180,E1 -10108.07,E2 -10108.07} C_VEL
LIN {X 0,Y 418.228,Z 191.388,A -85,B 0,C 180,E1 -10111.02,E2 -10111.02} C_VEL
LIN {X 0,Y 418.237,Z 191.386,A -85,B 0,C 180,E1 -10113.678,E2 -10113.678} C_VEL
LIN {X 0,Y 418.228,Z 191.389,A -85,B 0,C 180,E1 -10117.225,E2 -10117.225} C_VEL
LIN {X 0,Y 418.204,Z 191.382,A -85,B 0,C 180,E1 -10120.869,E2 -10120.869} C_VEL
LIN {X 0,Y 418.2,Z 191.391,A -85,B 0,C 180,E1 -10123.73,E2 -10123.73} C_VEL
LIN {X 0,Y 418.202,Z 191.394,A -85,B 0,C 180,E1 -10126.45,E2 -10126.45} C_VEL
LIN {X 0,Y 418.216,Z 191.393,A -85,B 0,C 180,E1 -10129.132,E2 -10129.132} C_VEL
LIN {X 0,Y 418.242,Z 191.412,A -85,B 0,C 180,E1 -10132.165,E2 -10132.165} C_VEL
LIN {X 0,Y 420.978,Z 202.779,A -85,B 0,C 180,E1 -10135.418,E2 -10135.418} C_VEL
LIN {X 0,Y 423.608,Z 214.676,A -85,B 0,C 180,E1 -10138.494,E2 -10138.494} C_VEL
LIN {X 0,Y 423.855,Z 218.529,A -85,B 0,C 180,E1 -10139.406,E2 -10139.406} C_VEL
LIN {X 0,Y 422.137,Z 234.033,A -85,B 0,C 180,E1 -10142.754,E2 -10142.754} C_VEL
LIN {X 0,Y 420.542,Z 251.081,A -85,B 0,C 180,E1 -10146.356,E2 -10146.356} C_VEL
LIN {X 0,Y 419.301,Z 267.523,A -85,B 0,C 180,E1 -10149.823,E2 -10149.823} C_VEL
LIN {X 0,Y 418.346,Z 283.056,A -85,B 0,C 180,E1 -10153.175,E2 -10153.175} C_VEL
LIN {X 0,Y 420.25,Z 302.632,A -85,B 0,C 180,E1 -10153.765,E2 -10153.765} C_VEL
LIN {X 0,Y 420.753,Z 315.096,A -85,B 0,C 180,E1 -10154.314,E2 -10154.314} C_VEL
LIN {X 0,Y 420.118,Z 328.638,A -85,B 0,C 180,E1 -10155.097,E2 -10155.097} C_VEL
LIN {X 0,Y 419.579,Z 339.756,A -85,B 0,C 180,E1 -10155.945,E2 -10155.945} C_VEL
LIN {X 0,Y 418.934,Z 350.913,A -85,B 0,C 180,E1 -10157.012,E2 -10157.012} C_VEL
LIN {X 0,Y 418.419,Z 360.394,A -85,B 0,C 180,E1 -10158.128,E2 -10158.128} C_VEL
LIN {X 0,Y 417.922,Z 368.849,A -85,B 0,C 180,E1 -10159.341,E2 -10159.341} C_VEL
LIN {X 0,Y 417.581,Z 377.104,A -85,B 0,C 180,E1 -10160.801,E2 -10160.801} C_VEL
LIN {X 0,Y 417.348,Z 383.73,A -85,B 0,C 180,E1 -10162.259,E2 -10162.259} C_VEL
LIN {X 0,Y 417.208,Z 388.772,A -85,B 0,C 180,E1 -10163.656,E2 -10163.656} C_VEL
LIN {X 0,Y 417.25,Z 392.977,A -85,B 0,C 180,E1 -10165.17,E2 -10165.17} C_VEL
LIN {X 0,Y 417.203,Z 395.006,A -85,B 0,C 180,E1 -10166.138,E2 -10166.138} C_VEL
LIN {X 0,Y 417.275,Z 396.607,A -85,B 0,C 180,E1 -10167.105,E2 -10167.105} C_VEL
LIN {X 0,Y 417.246,Z 397.763,A -85,B 0,C 180,E1 -10168.071,E2 -10168.071} C_VEL
LIN {X 0,Y 417.292,Z 398.449,A -85,B 0,C 180,E1 -10169.036,E2 -10169.036} C_VEL
LIN {X 0,Y 417.283,Z 398.717,A -85,B 0,C 180,E1 -10170.001,E2 -10170.001} C_VEL
LIN {X 0,Y 417.276,Z 398.574,A -85,B 0,C 180,E1 -10170.966,E2 -10170.966} C_VEL
LIN {X 0,Y 417.239,Z 397.971,A -85,B 0,C 180,E1 -10171.932,E2 -10171.932} C_VEL
LIN {X 0,Y 417.281,Z 396.937,A -85,B 0,C 180,E1 -10172.897,E2 -10172.897} C_VEL
LIN {X 0,Y 417.2,Z 395.479,A -85,B 0,C 180,E1 -10173.865,E2 -10173.865} C_VEL
LIN {X 0,Y 417.249,Z 392.433,A -85,B 0,C 180,E1 -10175.317,E2 -10175.317} C_VEL
LIN {X 0,Y 417.266,Z 388.309,A -85,B 0,C 180,E1 -10176.772,E2 -10176.772} C_VEL
LIN {X 0,Y 417.487,Z 381.975,A -85,B 0,C 180,E1 -10178.472,E2 -10178.472} C_VEL
LIN {X 0,Y 417.821,Z 375.064,A -85,B 0,C 180,E1 -10179.929,E2 -10179.929} C_VEL
LIN {X 0,Y 418.336,Z 366.581,A -85,B 0,C 180,E1 -10181.386,E2 -10181.386} C_VEL
LIN {X 0,Y 419.022,Z 356.293,A -85,B 0,C 180,E1 -10182.799,E2 -10182.799} C_VEL
LIN {X 0,Y 419.642,Z 346.593,A -85,B 0,C 180,E1 -10183.895,E2 -10183.895} C_VEL
LIN {X 0,Y 420.527,Z 335.757,A -85,B 0,C 180,E1 -10184.89,E2 -10184.89} C_VEL
LIN {X 0,Y 421.465,Z 322.587,A -85,B 0,C 180,E1 -10185.847,E2 -10185.847} C_VEL
LIN {X 0,Y 421.835,Z 312.202,A -85,B 0,C 180,E1 -10186.454,E2 -10186.454} C_VEL
LIN {X 0,Y 421.282,Z 298.896,A -85,B 0,C 180,E1 -10187.094,E2 -10187.094} C_VEL
LIN {X 0,Y 419.304,Z 282.822,A -85,B 0,C 180,E1 -10187.722,E2 -10187.722} C_VEL
LIN {X 0,Y 418.646,Z 278.074,A -85,B 0,C 180,E1 -10187.905,E2 -10187.905} C_VEL
LIN {X 0,Y 419.882,Z 259.522,A -85,B 0,C 180,E1 -10191.866,E2 -10191.866} C_VEL
LIN {X 0,Y 421.439,Z 240.929,A -85,B 0,C 180,E1 -10195.774,E2 -10195.774} C_VEL
LIN {X 0,Y 423.156,Z 224.235,A -85,B 0,C 180,E1 -10199.338,E2 -10199.338} C_VEL
LIN {X 0,Y 423.903,Z 216.992,A -85,B 0,C 180,E1 -10200.929,E2 -10200.929} C_VEL
LIN {X 0,Y 422.488,Z 209.775,A -85,B 0,C 180,E1 -10202.728,E2 -10202.728} C_VEL
LIN {X 0,Y 420.297,Z 199.924,A -85,B 0,C 180,E1 -10205.356,E2 -10205.356} C_VEL
LIN {X 0,Y 418.243,Z 191.389,A -85,B 0,C 180,E1 -10207.836,E2 -10207.836} C_VEL
LIN {X 0,Y 418.227,Z 191.389,A -85,B 0,C 180,E1 -10210.949,E2 -10210.949} C_VEL
LIN {X 0,Y 418.215,Z 191.391,A -85,B 0,C 180,E1 -10213.73,E2 -10213.73} C_VEL
LIN {X 0,Y 418.214,Z 191.391,A -85,B 0,C 180,E1 -10216.449,E2 -10216.449} C_VEL
LIN {X 0,Y 418.259,Z 191.505,A -85,B 0,C 180,E1 -10219.056,E2 -10219.056} C_VEL
LIN {X 0,Y 419.802,Z 197.517,A -85,B 0,C 180,E1 -10221.892,E2 -10221.892} C_VEL
LIN {X 0,Y 420.914,Z 202.916,A -85,B 0,C 180,E1 -10224.24,E2 -10224.24} C_VEL
LIN {X 0,Y 420.933,Z 207.342,A -85,B 0,C 180,E1 -10225.991,E2 -10225.991} C_VEL
LIN {X 0,Y 420.185,Z 217.395,A -85,B 0,C 180,E1 -10229.882,E2 -10229.882} C_VEL
LIN {X 0,Y 419.896,Z 224.212,A -85,B 0,C 180,E1 -10232.511,E2 -10232.511} C_VEL
LIN {X 0,Y 419.7,Z 230.076,A -85,B 0,C 180,E1 -10234.724,E2 -10234.724} C_VEL
LIN {X 0,Y 419.369,Z 238.08,A -85,B 0,C 180,E1 -10237.848,E2 -10237.848} C_VEL
LIN {X 0,Y 419.107,Z 245.95,A -85,B 0,C 180,E1 -10240.913,E2 -10240.913} C_VEL
LIN {X 0,Y 419.026,Z 249.417,A -85,B 0,C 180,E1 -10242.23,E2 -10242.23} C_VEL
LIN {X 0,Y 422.566,Z 262.137,A -85,B 0,C 180,E1 -10242.939,E2 -10242.939} C_VEL
LIN {X 0,Y 423.54,Z 267.786,A -85,B 0,C 180,E1 -10243.276,E2 -10243.276} C_VEL
LIN {X 0,Y 422.881,Z 279.834,A -85,B 0,C 180,E1 -10243.961,E2 -10243.961} C_VEL
LIN {X 0,Y 422.172,Z 291.057,A -85,B 0,C 180,E1 -10244.777,E2 -10244.777} C_VEL
LIN {X 0,Y 421.374,Z 301.801,A -85,B 0,C 180,E1 -10245.758,E2 -10245.758} C_VEL
LIN {X 0,Y 420.469,Z 312.524,A -85,B 0,C 180,E1 -10246.959,E2 -10246.959} C_VEL
LIN {X 0,Y 419.725,Z 321.248,A -85,B 0,C 180,E1 -10248.164,E2 -10248.164} C_VEL
LIN {X 0,Y 419.07,Z 329.766,A -85,B 0,C 180,E1 -10249.614,E2 -10249.614} C_VEL
LIN {X 0,Y 418.481,Z 336.686,A -85,B 0,C 180,E1 -10251.063,E2 -10251.063} C_VEL
LIN {X 0,Y 418.091,Z 341.354,A -85,B 0,C 180,E1 -10252.272,E2 -10252.272} C_VEL
LIN {X 0,Y 417.711,Z 345.869,A -85,B 0,C 180,E1 -10253.721,E2 -10253.721} C_VEL
LIN {X 0,Y 417.613,Z 349.269,A -85,B 0,C 180,E1 -10255.173,E2 -10255.173} C_VEL
LIN {X 0,Y 417.464,Z 350.984,A -85,B 0,C 180,E1 -10256.139,E2 -10256.139} C_VEL
LIN {X 0,Y 417.335,Z 352.249,A -85,B 0,C 180,E1 -10257.104,E2 -10257.104} C_VEL
LIN {X 0,Y 417.239,Z 353.117,A -85,B 0,C 180,E1 -10258.069,E2 -10258.069} C_VEL
LIN {X 0,Y 417.16,Z 353.584,A -85,B 0,C 180,E1 -10259.035,E2 -10259.035} C_VEL
LIN {X 0,Y 417.114,Z 353.602,A -85,B 0,C 180,E1 -10260,E2 -10260} C_VEL
LIN {X 0,Y 417.163,Z 352.442,A -85,B 0,C 180,E1 -10261.931,E2 -10261.931} C_VEL
LIN {X 0,Y 417.283,Z 351.223,A -85,B 0,C 180,E1 -10262.896,E2 -10262.896} C_VEL
LIN {X 0,Y 417.296,Z 348.603,A -85,B 0,C 180,E1 -10264.347,E2 -10264.347} C_VEL
LIN {X 0,Y 417.541,Z 343.917,A -85,B 0,C 180,E1 -10266.139,E2 -10266.139} C_VEL
LIN {X 0,Y 417.77,Z 338.309,A -85,B 0,C 180,E1 -10267.734,E2 -10267.734} C_VEL
LIN {X 0,Y 418.156,Z 331.772,A -85,B 0,C 180,E1 -10269.188,E2 -10269.188} C_VEL
LIN {X 0,Y 418.634,Z 323.668,A -85,B 0,C 180,E1 -10270.642,E2 -10270.642} C_VEL
LIN {X 0,Y 419.132,Z 315.425,A -85,B 0,C 180,E1 -10271.853,E2 -10271.853} C_VEL
LIN {X 0,Y 419.777,Z 305.365,A -85,B 0,C 180,E1 -10273.063,E2 -10273.063} C_VEL
LIN {X 0,Y 420.382,Z 293.406,A -85,B 0,C 180,E1 -10274.225,E2 -10274.225} C_VEL
LIN {X 0,Y 420.994,Z 281.625,A -85,B 0,C 180,E1 -10275.12,E2 -10275.12} C_VEL
LIN {X 0,Y 421.648,Z 268.271,A -85,B 0,C 180,E1 -10275.901,E2 -10275.901} C_VEL
LIN {X 0,Y 421.287,Z 263.021,A -85,B 0,C 180,E1 -10276.164,E2 -10276.164} C_VEL
LIN {X 0,Y 418.71,Z 249.135,A -85,B 0,C 180,E1 -10276.753,E2 -10276.753} C_VEL
LIN {X 0,Y 418.154,Z 246.111,A -85,B 0,C 180,E1 -10276.879,E2 -10276.879} C_VEL
LIN {X 0,Y 418.29,Z 237.57,A -85,B 0,C 180,E1 -10280.162,E2 -10280.162} C_VEL
LIN {X 0,Y 418.5,Z 229.597,A -85,B 0,C 180,E1 -10283.244,E2 -10283.244} C_VEL
LIN {X 0,Y 418.68,Z 221.448,A -85,B 0,C 180,E1 -10286.413,E2 -10286.413} C_VEL
LIN {X 0,Y 418.954,Z 213.028,A -85,B 0,C 180,E1 -10289.685,E2 -10289.685} C_VEL
LIN {X 0,Y 419.137,Z 205.947,A -85,B 0,C 180,E1 -10292.451,E2 -10292.451} C_VEL
LIN {X 0,Y 419.262,Z 198.509,A -85,B 0,C 180,E1 -10295.332,E2 -10295.332} C_VEL
LIN {X 0,Y 418.729,Z 193.96,A -85,B 0,C 180,E1 -10297.174,E2 -10297.174} C_VEL
LIN {X 0,Y 418.275,Z 191.384,A -85,B 0,C 180,E1 -10298.277,E2 -10298.277} C_VEL
LIN {X 0,Y 418.225,Z 191.392,A -85,B 0,C 180,E1 -10300.948,E2 -10300.948} C_VEL
LIN {X 0,Y 418.214,Z 191.39,A -85,B 0,C 180,E1 -10303.729,E2 -10303.729} C_VEL
LIN {X 0,Y 418.214,Z 191.39,A -85,B 0,C 180,E1 -10306.448,E2 -10306.448} C_VEL
LIN {X 0,Y 418.225,Z 191.391,A -85,B 0,C 180,E1 -10309.13,E2 -10309.13} C_VEL
LIN {X 0,Y 418.224,Z 191.393,A -85,B 0,C 180,E1 -10312.168,E2 -10312.168} C_VEL
LIN {X 0,Y 418.257,Z 191.389,A -85,B 0,C 180,E1 -10315.422,E2 -10315.422} C_VEL
LIN {X 0,Y 418.187,Z 191.397,A -85,B 0,C 180,E1 -10318.601,E2 -10318.601} C_VEL
LIN {X 0,Y 418.065,Z 191.412,A -85,B 0,C 180,E1 -10320.946,E2 -10320.946} C_VEL
LIN {X 0,Y 418.024,Z 195.002,A -85,B 0,C 180,E1 -10324.078,E2 -10324.078} C_VEL
LIN {X 0,Y 417.92,Z 198.865,A -85,B 0,C 180,E1 -10327.244,E2 -10327.244} C_VEL
LIN {X 0,Y 417.857,Z 202.762,A -85,B 0,C 180,E1 -10330.369,E2 -10330.369} C_VEL
LIN {X 0,Y 417.833,Z 206.839,A -85,B 0,C 180,E1 -10333.486,E2 -10333.486} C_VEL
LIN {X 0,Y 417.895,Z 212.308,A -85,B 0,C 180,E1 -10337.37,E2 -10337.37} C_VEL
LIN {X 0,Y 417.833,Z 214.745,A -85,B 0,C 180,E1 -10338.969,E2 -10338.969} C_VEL
LIN {X 0,Y 420.371,Z 225.96,A -85,B 0,C 180,E1 -10339.536,E2 -10339.536} C_VEL
LIN {X 0,Y 420.891,Z 229.443,A -85,B 0,C 180,E1 -10339.749,E2 -10339.749} C_VEL
LIN {X 0,Y 420.744,Z 238.387,A -85,B 0,C 180,E1 -10340.383,E2 -10340.383} C_VEL
LIN {X 0,Y 420.379,Z 246.653,A -85,B 0,C 180,E1 -10341.17,E2 -10341.17} C_VEL
LIN {X 0,Y 419.97,Z 253.706,A -85,B 0,C 180,E1 -10342.063,E2 -10342.063} C_VEL
LIN {X 0,Y 419.805,Z 258.322,A -85,B 0,C 180,E1 -10342.786,E2 -10342.786} C_VEL
LIN {X 0,Y 419.435,Z 263.232,A -85,B 0,C 180,E1 -10343.746,E2 -10343.746} C_VEL
LIN {X 0,Y 419.071,Z 267.071,A -85,B 0,C 180,E1 -10344.706,E2 -10344.706} C_VEL
LIN {X 0,Y 418.996,Z 270.021,A -85,B 0,C 180,E1 -10345.67,E2 -10345.67} C_VEL
LIN {X 0,Y 418.473,Z 273.184,A -85,B 0,C 180,E1 -10347.111,E2 -10347.111} C_VEL
LIN {X 0,Y 418.442,Z 273.792,A -85,B 0,C 180,E1 -10347.558,E2 -10347.558} C_VEL
LIN {X 0,Y 417.737,Z 274.862,A -85,B 0,C 180,E1 -10348.35,E2 -10348.35} C_VEL
LIN {X 0,Y 414.809,Z 275.973,A -85,B 0,C 180,E1 -10349.644,E2 -10349.644} C_VEL
LIN {X 0,Y 411.952,Z 276.203,A -85,B 0,C 180,E1 -10350.961,E2 -10350.961} C_VEL
LIN {X 0,Y 411.371,Z 275.697,A -85,B 0,C 180,E1 -10351.778,E2 -10351.778} C_VEL
LIN {X 0,Y 411.454,Z 274.319,A -85,B 0,C 180,E1 -10352.936,E2 -10352.936} C_VEL
LIN {X 0,Y 411.988,Z 271.265,A -85,B 0,C 180,E1 -10354.401,E2 -10354.401} C_VEL
LIN {X 0,Y 412.115,Z 266.672,A -85,B 0,C 180,E1 -10355.872,E2 -10355.872} C_VEL
LIN {X 0,Y 412.517,Z 263.599,A -85,B 0,C 180,E1 -10356.602,E2 -10356.602} C_VEL
LIN {X 0,Y 412.906,Z 257.104,A -85,B 0,C 180,E1 -10357.825,E2 -10357.825} C_VEL
LIN {X 0,Y 413.387,Z 250.079,A -85,B 0,C 180,E1 -10358.8,E2 -10358.8} C_VEL
LIN {X 0,Y 413.644,Z 244.185,A -85,B 0,C 180,E1 -10359.454,E2 -10359.454} C_VEL
LIN {X 0,Y 413.933,Z 237.157,A -85,B 0,C 180,E1 -10360.082,E2 -10360.082} C_VEL
LIN {X 0,Y 413.918,Z 229.159,A -85,B 0,C 180,E1 -10360.627,E2 -10360.627} C_VEL
LIN {X 0,Y 411.611,Z 218.843,A -85,B 0,C 180,E1 -10361.201,E2 -10361.201} C_VEL
LIN {X 0,Y 410.831,Z 215.36,A -85,B 0,C 180,E1 -10361.376,E2 -10361.376} C_VEL
LIN {X 0,Y 410.764,Z 211.664,A -85,B 0,C 180,E1 -10363.858,E2 -10363.858} C_VEL
LIN {X 0,Y 410.8,Z 207.43,A -85,B 0,C 180,E1 -10366.907,E2 -10366.907} C_VEL
LIN {X 0,Y 410.809,Z 203.431,A -85,B 0,C 180,E1 -10370.007,E2 -10370.007} C_VEL
LIN {X 0,Y 410.901,Z 199.511,A -85,B 0,C 180,E1 -10373.164,E2 -10373.164} C_VEL
LIN {X 0,Y 410.984,Z 195.535,A -85,B 0,C 180,E1 -10376.397,E2 -10376.397} C_VEL
LIN {X 0,Y 411.05,Z 192.286,A -85,B 0,C 180,E1 -10379.31,E2 -10379.31} C_VEL
LIN {X 0,Y 411.152,Z 192.271,A -85,B 0,C 180,E1 -10381.997,E2 -10381.997} C_VEL
LIN {X 0,Y 411.207,Z 192.264,A -85,B 0,C 180,E1 -10384.877,E2 -10384.877} C_VEL
LIN {X 0,Y 411.205,Z 192.262,A -85,B 0,C 180,E1 -10388.168,E2 -10388.168} C_VEL
LIN {X 0,Y 411.159,Z 192.271,A -85,B 0,C 180,E1 -10391.227,E2 -10391.227} C_VEL
LIN {X 0,Y 411.173,Z 192.265,A -85,B 0,C 180,E1 -10394.489,E2 -10394.489} C_VEL
LIN {X 0,Y 411.17,Z 192.267,A -85,B 0,C 180,E1 -10398.193,E2 -10398.193} C_VEL
LIN {X 0,Y 411.218,Z 192.265,A -85,B 0,C 180,E1 -10400.776,E2 -10400.776} C_VEL
LIN {X 0,Y 411.191,Z 192.267,A -85,B 0,C 180,E1 -10404.47,E2 -10404.47} C_VEL
LIN {X 0,Y 411.163,Z 192.267,A -85,B 0,C 180,E1 -10408.002,E2 -10408.002} C_VEL
LIN {X 0,Y 411.214,Z 192.257,A -85,B 0,C 180,E1 -10411.409,E2 -10411.409} C_VEL
LIN {X 0,Y 411.226,Z 192.253,A -85,B 0,C 180,E1 -10414.706,E2 -10414.706} C_VEL
LIN {X 0,Y 411.195,Z 192.267,A -85,B 0,C 180,E1 -10417.913,E2 -10417.913} C_VEL
LIN {X 0,Y 411.214,Z 192.258,A -85,B 0,C 180,E1 -10421.051,E2 -10421.051} C_VEL
LIN {X 0,Y 411.252,Z 192.25,A -85,B 0,C 180,E1 -10424.131,E2 -10424.131} C_VEL
LIN {X 0,Y 411.292,Z 192.252,A -85,B 0,C 180,E1 -10427.165,E2 -10427.165} C_VEL
LIN {X 0,Y 411.283,Z 192.244,A -85,B 0,C 180,E1 -10430.161,E2 -10430.161} C_VEL
LIN {X 0,Y 411.44,Z 192.236,A -85,B 0,C 180,E1 -10433.133,E2 -10433.133} C_VEL
LIN {X 0,Y 411.298,Z 192.246,A -85,B 0,C 180,E1 -10435.099,E2 -10435.099} C_VEL
LIN {X 0,Y 411.502,Z 192.223,A -85,B 0,C 180,E1 -10438.042,E2 -10438.042} C_VEL
LIN {X 0,Y 411.629,Z 192.2,A -85,B 0,C 180,E1 -10440,E2 -10440} C_VEL
LIN {X 0,Y 411.443,Z 192.234,A -85,B 0,C 180,E1 -10442.937,E2 -10442.937} C_VEL
LIN {X 0,Y 411.446,Z 192.235,A -85,B 0,C 180,E1 -10446.867,E2 -10446.867} C_VEL
LIN {X 0,Y 411.342,Z 192.241,A -85,B 0,C 180,E1 -10448.845,E2 -10448.845} C_VEL
LIN {X 0,Y 411.271,Z 192.254,A -85,B 0,C 180,E1 -10451.833,E2 -10451.833} C_VEL
LIN {X 0,Y 411.247,Z 192.258,A -85,B 0,C 180,E1 -10454.853,E2 -10454.853} C_VEL
LIN {X 0,Y 411.233,Z 192.256,A -85,B 0,C 180,E1 -10457.916,E2 -10457.916} C_VEL
LIN {X 0,Y 411.184,Z 192.265,A -85,B 0,C 180,E1 -10461.035,E2 -10461.035} C_VEL
LIN {X 0,Y 411.18,Z 192.269,A -85,B 0,C 180,E1 -10464.218,E2 -10464.218} C_VEL
LIN {X 0,Y 411.135,Z 192.275,A -85,B 0,C 180,E1 -10467.487,E2 -10467.487} C_VEL
LIN {X 0,Y 411.185,Z 192.27,A -85,B 0,C 180,E1 -10469.714,E2 -10469.714} C_VEL
LIN {X 0,Y 411.197,Z 192.266,A -85,B 0,C 180,E1 -10473.157,E2 -10473.157} C_VEL
LIN {X 0,Y 411.182,Z 192.266,A -85,B 0,C 180,E1 -10476.553,E2 -10476.553} C_VEL
LIN {X 0,Y 411.169,Z 192.263,A -85,B 0,C 180,E1 -10479.723,E2 -10479.723} C_VEL
LIN {X 0,Y 411.162,Z 192.271,A -85,B 0,C 180,E1 -10483.135,E2 -10483.135} C_VEL
LIN {X 0,Y 411.161,Z 192.269,A -85,B 0,C 180,E1 -10485.882,E2 -10485.882} C_VEL
LIN {X 0,Y 411.157,Z 192.266,A -85,B 0,C 180,E1 -10488.773,E2 -10488.773} C_VEL
LIN {X 0,Y 411.24,Z 192.385,A -85,B 0,C 180,E1 -10491.707,E2 -10491.707} C_VEL
LIN {X 0,Y 413.932,Z 203.686,A -85,B 0,C 180,E1 -10495.04,E2 -10495.04} C_VEL
LIN {X 0,Y 416.447,Z 215.045,A -85,B 0,C 180,E1 -10498.061,E2 -10498.061} C_VEL
LIN {X 0,Y 417.073,Z 218.663,A -85,B 0,C 180,E1 -10498.966,E2 -10498.966} C_VEL
LIN {X 0,Y 415.329,Z 233.568,A -85,B 0,C 180,E1 -10502.269,E2 -10502.269} C_VEL
LIN {X 0,Y 413.682,Z 250.491,A -85,B 0,C 180,E1 -10505.939,E2 -10505.939} C_VEL
LIN {X 0,Y 412.415,Z 266.513,A -85,B 0,C 180,E1 -10509.406,E2 -10509.406} C_VEL
LIN {X 0,Y 411.319,Z 282.55,A -85,B 0,C 180,E1 -10512.943,E2 -10512.943} C_VEL
LIN {X 0,Y 413.191,Z 301.715,A -85,B 0,C 180,E1 -10513.528,E2 -10513.528} C_VEL
LIN {X 0,Y 413.792,Z 314.673,A -85,B 0,C 180,E1 -10514.107,E2 -10514.107} C_VEL
LIN {X 0,Y 413.24,Z 327.264,A -85,B 0,C 180,E1 -10514.843,E2 -10514.843} C_VEL
LIN {X 0,Y 412.592,Z 338.608,A -85,B 0,C 180,E1 -10515.702,E2 -10515.702} C_VEL
LIN {X 0,Y 411.913,Z 350.454,A -85,B 0,C 180,E1 -10516.848,E2 -10516.848} C_VEL
LIN {X 0,Y 411.387,Z 359.465,A -85,B 0,C 180,E1 -10517.922,E2 -10517.922} C_VEL
LIN {X 0,Y 410.903,Z 368.045,A -85,B 0,C 180,E1 -10519.157,E2 -10519.157} C_VEL
LIN {X 0,Y 410.537,Z 376.372,A -85,B 0,C 180,E1 -10520.642,E2 -10520.642} C_VEL
LIN {X 0,Y 410.278,Z 383.06,A -85,B 0,C 180,E1 -10522.125,E2 -10522.125} C_VEL
LIN {X 0,Y 410.137,Z 388.518,A -85,B 0,C 180,E1 -10523.656,E2 -10523.656} C_VEL
LIN {X 0,Y 410.177,Z 392.432,A -85,B 0,C 180,E1 -10525.087,E2 -10525.087} C_VEL
LIN {X 0,Y 410.112,Z 394.491,A -85,B 0,C 180,E1 -10526.071,E2 -10526.071} C_VEL
LIN {X 0,Y 410.203,Z 396.115,A -85,B 0,C 180,E1 -10527.055,E2 -10527.055} C_VEL
LIN {X 0,Y 410.167,Z 397.301,A -85,B 0,C 180,E1 -10528.037,E2 -10528.037} C_VEL
LIN {X 0,Y 410.214,Z 398.018,A -85,B 0,C 180,E1 -10529.02,E2 -10529.02} C_VEL
LIN {X 0,Y 410.221,Z 398.306,A -85,B 0,C 180,E1 -10530.001,E2 -10530.001} C_VEL
LIN {X 0,Y 410.186,Z 398.179,A -85,B 0,C 180,E1 -10530.983,E2 -10530.983} C_VEL
LIN {X 0,Y 410.162,Z 397.613,A -85,B 0,C 180,E1 -10531.965,E2 -10531.965} C_VEL
LIN {X 0,Y 410.19,Z 396.594,A -85,B 0,C 180,E1 -10532.948,E2 -10532.948} C_VEL
LIN {X 0,Y 410.108,Z 395.154,A -85,B 0,C 180,E1 -10533.932,E2 -10533.932} C_VEL
LIN {X 0,Y 410.155,Z 392.146,A -85,B 0,C 180,E1 -10535.409,E2 -10535.409} C_VEL
LIN {X 0,Y 410.191,Z 388.059,A -85,B 0,C 180,E1 -10536.89,E2 -10536.89} C_VEL
LIN {X 0,Y 410.444,Z 381.804,A -85,B 0,C 180,E1 -10538.618,E2 -10538.618} C_VEL
LIN {X 0,Y 410.837,Z 373.688,A -85,B 0,C 180,E1 -10540.349,E2 -10540.349} C_VEL
LIN {X 0,Y 411.517,Z 364.959,A -85,B 0,C 180,E1 -10541.827,E2 -10541.827} C_VEL
LIN {X 0,Y 412.177,Z 355.057,A -85,B 0,C 180,E1 -10543.192,E2 -10543.192} C_VEL
LIN {X 0,Y 412.904,Z 345.367,A -85,B 0,C 180,E1 -10544.29,E2 -10544.29} C_VEL
LIN {X 0,Y 413.953,Z 333.329,A -85,B 0,C 180,E1 -10545.385,E2 -10545.385} C_VEL
LIN {X 0,Y 414.835,Z 321.653,A -85,B 0,C 180,E1 -10546.234,E2 -10546.234} C_VEL
LIN {X 0,Y 415.163,Z 313.51,A -85,B 0,C 180,E1 -10546.726,E2 -10546.726} C_VEL
LIN {X 0,Y 414.73,Z 300.216,A -85,B 0,C 180,E1 -10547.415,E2 -10547.415} C_VEL
LIN {X 0,Y 412.886,Z 284.405,A -85,B 0,C 180,E1 -10548.073,E2 -10548.073} C_VEL
LIN {X 0,Y 411.675,Z 276.438,A -85,B 0,C 180,E1 -10548.431,E2 -10548.431} C_VEL
LIN {X 0,Y 412.991,Z 258.861,A -85,B 0,C 180,E1 -10552.25,E2 -10552.25} C_VEL
LIN {X 0,Y 414.569,Z 240.757,A -85,B 0,C 180,E1 -10556.154,E2 -10556.154} C_VEL
LIN {X 0,Y 416.307,Z 225.043,A -85,B 0,C 180,E1 -10559.591,E2 -10559.591} C_VEL
LIN {X 0,Y 417.048,Z 218.599,A -85,B 0,C 180,E1 -10561.035,E2 -10561.035} C_VEL
LIN {X 0,Y 415.153,Z 209.473,A -85,B 0,C 180,E1 -10563.381,E2 -10563.381} C_VEL
LIN {X 0,Y 413.062,Z 200.193,A -85,B 0,C 180,E1 -10565.945,E2 -10565.945} C_VEL
LIN {X 0,Y 411.213,Z 192.266,A -85,B 0,C 180,E1 -10568.332,E2 -10568.332} C_VEL
LIN {X 0,Y 411.182,Z 192.268,A -85,B 0,C 180,E1 -10571.806,E2 -10571.806} C_VEL
LIN {X 0,Y 411.181,Z 192.268,A -85,B 0,C 180,E1 -10575.51,E2 -10575.51} C_VEL
LIN {X 0,Y 411.227,Z 192.326,A -85,B 0,C 180,E1 -10577.789,E2 -10577.789} C_VEL
LIN {X 0,Y 412.807,Z 198.384,A -85,B 0,C 180,E1 -10580.956,E2 -10580.956} C_VEL
LIN {X 0,Y 413.988,Z 203.961,A -85,B 0,C 180,E1 -10583.546,E2 -10583.546} C_VEL
LIN {X 0,Y 414.338,Z 206.799,A -85,B 0,C 180,E1 -10584.781,E2 -10584.781} C_VEL
LIN {X 0,Y 413.957,Z 212.601,A -85,B 0,C 180,E1 -10587.092,E2 -10587.092} C_VEL
LIN {X 0,Y 413.258,Z 222.439,A -85,B 0,C 180,E1 -10591.008,E2 -10591.008} C_VEL
LIN {X 0,Y 412.862,Z 231.29,A -85,B 0,C 180,E1 -10594.45,E2 -10594.45} C_VEL
LIN {X 0,Y 412.532,Z 238.915,A -85,B 0,C 180,E1 -10597.461,E2 -10597.461} C_VEL
LIN {X 0,Y 412.182,Z 248.105,A -85,B 0,C 180,E1 -10601.097,E2 -10601.097} C_VEL
LIN {X 0,Y 412.1,Z 249.83,A -85,B 0,C 180,E1 -10601.776,E2 -10601.776} C_VEL
LIN {X 0,Y 415.516,Z 261.516,A -85,B 0,C 180,E1 -10602.465,E2 -10602.465} C_VEL
LIN {X 0,Y 416.963,Z 268.642,A -85,B 0,C 180,E1 -10602.919,E2 -10602.919} C_VEL
LIN {X 0,Y 416.22,Z 281.752,A -85,B 0,C 180,E1 -10603.697,E2 -10603.697} C_VEL
LIN {X 0,Y 415.364,Z 293.709,A -85,B 0,C 180,E1 -10604.625,E2 -10604.625} C_VEL
LIN {X 0,Y 414.428,Z 305.398,A -85,B 0,C 180,E1 -10605.765,E2 -10605.765} C_VEL
LIN {X 0,Y 413.443,Z 315.445,A -85,B 0,C 180,E1 -10606.983,E2 -10606.983} C_VEL
LIN {X 0,Y 412.671,Z 323.719,A -85,B 0,C 180,E1 -10608.208,E2 -10608.208} C_VEL
LIN {X 0,Y 412.077,Z 331.86,A -85,B 0,C 180,E1 -10609.684,E2 -10609.684} C_VEL
LIN {X 0,Y 411.417,Z 338.409,A -85,B 0,C 180,E1 -10611.156,E2 -10611.156} C_VEL
LIN {X 0,Y 410.967,Z 343.833,A -85,B 0,C 180,E1 -10612.693,E2 -10612.693} C_VEL
LIN {X 0,Y 410.504,Z 347.725,A -85,B 0,C 180,E1 -10614.104,E2 -10614.104} C_VEL
LIN {X 0,Y 410.568,Z 349.843,A -85,B 0,C 180,E1 -10615.09,E2 -10615.09} C_VEL
LIN {X 0,Y 410.417,Z 351.507,A -85,B 0,C 180,E1 -10616.072,E2 -10616.072} C_VEL
LIN {X 0,Y 410.163,Z 353.587,A -85,B 0,C 180,E1 -10618.036,E2 -10618.036} C_VEL
LIN {X 0,Y 410.078,Z 354.012,A -85,B 0,C 180,E1 -10619.018,E2 -10619.018} C_VEL
LIN {X 0,Y 410.031,Z 353.997,A -85,B 0,C 180,E1 -10620,E2 -10620} C_VEL
LIN {X 0,Y 410.036,Z 353.586,A -85,B 0,C 180,E1 -10620.982,E2 -10620.982} C_VEL
LIN {X 0,Y 410.091,Z 352.777,A -85,B 0,C 180,E1 -10621.964,E2 -10621.964} C_VEL
LIN {X 0,Y 410.217,Z 351.509,A -85,B 0,C 180,E1 -10622.946,E2 -10622.946} C_VEL
LIN {X 0,Y 410.21,Z 348.832,A -85,B 0,C 180,E1 -10624.422,E2 -10624.422} C_VEL
LIN {X 0,Y 410.398,Z 345.113,A -85,B 0,C 180,E1 -10625.898,E2 -10625.898} C_VEL
LIN {X 0,Y 410.612,Z 340.256,A -85,B 0,C 180,E1 -10627.375,E2 -10627.375} C_VEL
LIN {X 0,Y 410.968,Z 334.125,A -85,B 0,C 180,E1 -10628.854,E2 -10628.854} C_VEL
LIN {X 0,Y 411.424,Z 326.518,A -85,B 0,C 180,E1 -10630.333,E2 -10630.333} C_VEL
LIN {X 0,Y 412.018,Z 316.986,A -85,B 0,C 180,E1 -10631.811,E2 -10631.811} C_VEL
LIN {X 0,Y 412.682,Z 307.25,A -85,B 0,C 180,E1 -10633.041,E2 -10633.041} C_VEL
LIN {X 0,Y 413.257,Z 296.572,A -85,B 0,C 180,E1 -10634.135,E2 -10634.135} C_VEL
LIN {X 0,Y 413.929,Z 284.418,A -85,B 0,C 180,E1 -10635.132,E2 -10635.132} C_VEL
LIN {X 0,Y 414.529,Z 272.02,A -85,B 0,C 180,E1 -10635.916,E2 -10635.916} C_VEL
LIN {X 0,Y 414.549,Z 265.255,A -85,B 0,C 180,E1 -10636.269,E2 -10636.269} C_VEL
LIN {X 0,Y 412.127,Z 251.972,A -85,B 0,C 180,E1 -10636.884,E2 -10636.884} C_VEL
LIN {X 0,Y 411.113,Z 246.463,A -85,B 0,C 180,E1 -10637.087,E2 -10637.087} C_VEL
LIN {X 0,Y 411.266,Z 237.634,A -85,B 0,C 180,E1 -10640.507,E2 -10640.507} C_VEL
LIN {X 0,Y 411.486,Z 229.524,A -85,B 0,C 180,E1 -10643.664,E2 -10643.664} C_VEL
LIN {X 0,Y 411.735,Z 221.282,A -85,B 0,C 180,E1 -10646.887,E2 -10646.887} C_VEL
LIN {X 0,Y 412.076,Z 211.366,A -85,B 0,C 180,E1 -10650.774,E2 -10650.774} C_VEL
LIN {X 0,Y 412.239,Z 202.545,A -85,B 0,C 180,E1 -10654.236,E2 -10654.236} C_VEL
LIN {X 0,Y 412.167,Z 198.039,A -85,B 0,C 180,E1 -10656.035,E2 -10656.035} C_VEL
LIN {X 0,Y 411.265,Z 192.257,A -85,B 0,C 180,E1 -10658.446,E2 -10658.446} C_VEL
LIN {X 0,Y 411.178,Z 192.267,A -85,B 0,C 180,E1 -10661.806,E2 -10661.806} C_VEL
LIN {X 0,Y 411.181,Z 192.265,A -85,B 0,C 180,E1 -10665.509,E2 -10665.509} C_VEL
LIN {X 0,Y 411.167,Z 192.27,A -85,B 0,C 180,E1 -10668.772,E2 -10668.772} C_VEL
LIN {X 0,Y 411.19,Z 192.269,A -85,B 0,C 180,E1 -10672.025,E2 -10672.025} C_VEL
LIN {X 0,Y 411.197,Z 192.269,A -85,B 0,C 180,E1 -10675.664,E2 -10675.664} C_VEL
LIN {X 0,Y 411.16,Z 192.272,A -85,B 0,C 180,E1 -10678.722,E2 -10678.722} C_VEL
LIN {X 0,Y 411.055,Z 192.285,A -85,B 0,C 180,E1 -10680.689,E2 -10680.689} C_VEL
LIN {X 0,Y 411.01,Z 194.123,A -85,B 0,C 180,E1 -10682.503,E2 -10682.503} C_VEL
LIN {X 0,Y 410.936,Z 198.029,A -85,B 0,C 180,E1 -10685.765,E2 -10685.765} C_VEL
LIN {X 0,Y 410.834,Z 201.967,A -85,B 0,C 180,E1 -10688.945,E2 -10688.945} C_VEL
LIN {X 0,Y 410.776,Z 205.926,A -85,B 0,C 180,E1 -10692.062,E2 -10692.062} C_VEL
LIN {X 0,Y 410.748,Z 210.084,A -85,B 0,C 180,E1 -10695.127,E2 -10695.127} C_VEL
LIN {X 0,Y 410.836,Z 214.474,A -85,B 0,C 180,E1 -10698.153,E2 -10698.153} C_VEL
LIN {X 0,Y 410.836,Z 215.39,A -85,B 0,C 180,E1 -10698.747,E2 -10698.747} C_VEL
LIN {X 0,Y 413.272,Z 226.269,A -85,B 0,C 180,E1 -10699.286,E2 -10699.286} C_VEL
LIN {X 0,Y 413.992,Z 230.878,A -85,B 0,C 180,E1 -10699.577,E2 -10699.577} C_VEL
LIN {X 0,Y 413.782,Z 241.033,A -85,B 0,C 180,E1 -10700.339,E2 -10700.339} C_VEL
LIN {X 0,Y 413.46,Z 247.713,A -85,B 0,C 180,E1 -10701.012,E2 -10701.012} C_VEL
LIN {X 0,Y 413.027,Z 254.792,A -85,B 0,C 180,E1 -10701.929,E2 -10701.929} C_VEL
LIN {X 0,Y 412.654,Z 260.713,A -85,B 0,C 180,E1 -10702.906,E2 -10702.906} C_VEL
LIN {X 0,Y 412.334,Z 265.29,A -85,B 0,C 180,E1 -10703.884,E2 -10703.884} C_VEL
LIN {X 0,Y 412.067,Z 269.634,A -85,B 0,C 180,E1 -10705.107,E2 -10705.107} C_VEL
LIN {X 0,Y 411.81,Z 272.226,A -85,B 0,C 180,E1 -10706.084,E2 -10706.084} C_VEL
LIN {X 0,Y 411.459,Z 274.164,A -85,B 0,C 180,E1 -10707.062,E2 -10707.062} C_VEL
LIN {X 0,Y 411.418,Z 275.467,A -85,B 0,C 180,E1 -10708.041,E2 -10708.041} C_VEL
LIN {X 0,Y 411.3,Z 276.245,A -85,B 0,C 180,E1 -10709.02,E2 -10709.02} C_VEL
LIN {X 0,Y 411.251,Z 276.512,A -85,B 0,C 180,E1 -10709.999,E2 -10709.999} C_VEL
LIN {X 0,Y 411.294,Z 276.289,A -85,B 0,C 180,E1 -10710.978,E2 -10710.978} C_VEL
LIN {X 0,Y 411.371,Z 275.697,A -85,B 0,C 180,E1 -10711.778,E2 -10711.778} C_VEL
LIN {X 0,Y 410.844,Z 274.947,A -85,B 0,C 180,E1 -10712.593,E2 -10712.593} C_VEL
LIN {X 0,Y 409.424,Z 273.905,A -85,B 0,C 180,E1 -10713.387,E2 -10713.387} C_VEL
LIN {X 0,Y 406.059,Z 270.844,A -85,B 0,C 180,E1 -10714.939,E2 -10714.939} C_VEL
LIN {X 0,Y 405.166,Z 268.625,A -85,B 0,C 180,E1 -10715.708,E2 -10715.708} C_VEL
LIN {X 0,Y 405.124,Z 267.717,A -85,B 0,C 180,E1 -10715.962,E2 -10715.962} C_VEL
LIN {X 0,Y 405.539,Z 264.625,A -85,B 0,C 180,E1 -10716.716,E2 -10716.716} C_VEL
LIN {X 0,Y 405.959,Z 258.169,A -85,B 0,C 180,E1 -10717.959,E2 -10717.959} C_VEL
LIN {X 0,Y 406.463,Z 251.204,A -85,B 0,C 180,E1 -10718.951,E2 -10718.951} C_VEL
LIN {X 0,Y 406.734,Z 245.194,A -85,B 0,C 180,E1 -10719.634,E2 -10719.634} C_VEL
LIN {X 0,Y 407.093,Z 237.012,A -85,B 0,C 180,E1 -10720.365,E2 -10720.365} C_VEL
LIN {X 0,Y 407.03,Z 230.434,A -85,B 0,C 180,E1 -10720.821,E2 -10720.821} C_VEL
LIN {X 0,Y 404.783,Z 220.239,A -85,B 0,C 180,E1 -10721.412,E2 -10721.412} C_VEL
LIN {X 0,Y 403.792,Z 216.004,A -85,B 0,C 180,E1 -10721.608,E2 -10721.608} C_VEL
LIN {X 0,Y 403.734,Z 212.314,A -85,B 0,C 180,E1 -10724.104,E2 -10724.104} C_VEL
LIN {X 0,Y 403.772,Z 208.027,A -85,B 0,C 180,E1 -10727.21,E2 -10727.21} C_VEL
LIN {X 0,Y 403.783,Z 203.96,A -85,B 0,C 180,E1 -10730.37,E2 -10730.37} C_VEL
LIN {X 0,Y 403.877,Z 199.962,A -85,B 0,C 180,E1 -10733.591,E2 -10733.591} C_VEL
LIN {X 0,Y 403.966,Z 195.978,A -85,B 0,C 180,E1 -10736.892,E2 -10736.892} C_VEL
LIN {X 0,Y 403.999,Z 193.309,A -85,B 0,C 180,E1 -10739.148,E2 -10739.148} C_VEL
LIN {X 0,Y 404.117,Z 193.148,A -85,B 0,C 180,E1 -10741.552,E2 -10741.552} C_VEL
LIN {X 0,Y 404.181,Z 193.14,A -85,B 0,C 180,E1 -10745.015,E2 -10745.015} C_VEL
LIN {X 0,Y 404.153,Z 193.142,A -85,B 0,C 180,E1 -10748.755,E2 -10748.755} C_VEL
LIN {X 0,Y 404.118,Z 193.146,A -85,B 0,C 180,E1 -10751.599,E2 -10751.599} C_VEL
LIN {X 0,Y 404.142,Z 193.141,A -85,B 0,C 180,E1 -10754.521,E2 -10754.521} C_VEL
LIN {X 0,Y 404.129,Z 193.146,A -85,B 0,C 180,E1 -10757.294,E2 -10757.294} C_VEL
LIN {X 0,Y 404.161,Z 193.137,A -85,B 0,C 180,E1 -10759.954,E2 -10759.954} C_VEL
LIN {X 0,Y 404.132,Z 193.143,A -85,B 0,C 180,E1 -10763.123,E2 -10763.123} C_VEL
LIN {X 0,Y 404.136,Z 193.141,A -85,B 0,C 180,E1 -10766.187,E2 -10766.187} C_VEL
LIN {X 0,Y 404.146,Z 193.14,A -85,B 0,C 180,E1 -10769.715,E2 -10769.715} C_VEL
LIN {X 0,Y 404.185,Z 193.135,A -85,B 0,C 180,E1 -10773.122,E2 -10773.122} C_VEL
LIN {X 0,Y 404.167,Z 193.131,A -85,B 0,C 180,E1 -10775.334,E2 -10775.334} C_VEL
LIN {X 0,Y 404.128,Z 193.14,A -85,B 0,C 180,E1 -10778.58,E2 -10778.58} C_VEL
LIN {X 0,Y 404.2,Z 193.137,A -85,B 0,C 180,E1 -10781.761,E2 -10781.761} C_VEL
LIN {X 0,Y 404.2,Z 193.126,A -85,B 0,C 180,E1 -10784.882,E2 -10784.882} C_VEL
LIN {X 0,Y 404.246,Z 193.128,A -85,B 0,C 180,E1 -10787.958,E2 -10787.958} C_VEL
LIN {X 0,Y 404.393,Z 193.109,A -85,B 0,C 180,E1 -10792.129,E2 -10792.129} C_VEL
LIN {X 0,Y 404.407,Z 193.104,A -85,B 0,C 180,E1 -10794.015,E2 -10794.015} C_VEL
LIN {X 0,Y 404.471,Z 193.099,A -85,B 0,C 180,E1 -10798.008,E2 -10798.008} C_VEL
LIN {X 0,Y 404.599,Z 193.075,A -85,B 0,C 180,E1 -10800,E2 -10800} C_VEL
LIN {X 0,Y 404.401,Z 193.111,A -85,B 0,C 180,E1 -10802.989,E2 -10802.989} C_VEL
LIN {X 0,Y 404.397,Z 193.112,A -85,B 0,C 180,E1 -10806.987,E2 -10806.987} C_VEL
LIN {X 0,Y 404.245,Z 193.124,A -85,B 0,C 180,E1 -10810.012,E2 -10810.012} C_VEL
LIN {X 0,Y 404.255,Z 193.121,A -85,B 0,C 180,E1 -10813.212,E2 -10813.212} C_VEL
LIN {X 0,Y 404.204,Z 193.13,A -85,B 0,C 180,E1 -10817.007,E2 -10817.007} C_VEL
LIN {X 0,Y 404.152,Z 193.144,A -85,B 0,C 180,E1 -10820.352,E2 -10820.352} C_VEL
LIN {X 0,Y 404.138,Z 193.146,A -85,B 0,C 180,E1 -10823.577,E2 -10823.577} C_VEL
LIN {X 0,Y 404.092,Z 193.149,A -85,B 0,C 180,E1 -10826.885,E2 -10826.885} C_VEL
LIN {X 0,Y 404.133,Z 193.144,A -85,B 0,C 180,E1 -10830.286,E2 -10830.286} C_VEL
LIN {X 0,Y 404.134,Z 193.142,A -85,B 0,C 180,E1 -10833.813,E2 -10833.813} C_VEL
LIN {X 0,Y 404.125,Z 193.146,A -85,B 0,C 180,E1 -10836.876,E2 -10836.876} C_VEL
LIN {X 0,Y 404.109,Z 193.14,A -85,B 0,C 180,E1 -10840.076,E2 -10840.076} C_VEL
LIN {X 0,Y 404.141,Z 193.146,A -85,B 0,C 180,E1 -10843.084,E2 -10843.084} C_VEL
LIN {X 0,Y 404.141,Z 193.143,A -85,B 0,C 180,E1 -10845.927,E2 -10845.927} C_VEL
LIN {X 0,Y 404.111,Z 193.142,A -85,B 0,C 180,E1 -10848.636,E2 -10848.636} C_VEL
LIN {X 0,Y 404.197,Z 193.22,A -85,B 0,C 180,E1 -10851.21,E2 -10851.21} C_VEL
LIN {X 0,Y 407.031,Z 205.213,A -85,B 0,C 180,E1 -10854.819,E2 -10854.819} C_VEL
LIN {X 0,Y 409.476,Z 216.361,A -85,B 0,C 180,E1 -10857.857,E2 -10857.857} C_VEL
LIN {X 0,Y 410.176,Z 220.641,A -85,B 0,C 180,E1 -10858.949,E2 -10858.949} C_VEL
LIN {X 0,Y 408.194,Z 236.696,A -85,B 0,C 180,E1 -10862.578,E2 -10862.578} C_VEL
LIN {X 0,Y 406.453,Z 253.984,A -85,B 0,C 180,E1 -10866.41,E2 -10866.41} C_VEL
LIN {X 0,Y 404.945,Z 272.265,A -85,B 0,C 180,E1 -10870.484,E2 -10870.484} C_VEL
LIN {X 0,Y 404.303,Z 282.18,A -85,B 0,C 180,E1 -10872.708,E2 -10872.708} C_VEL
LIN {X 0,Y 406.137,Z 301.454,A -85,B 0,C 180,E1 -10873.311,E2 -10873.311} C_VEL
LIN {X 0,Y 406.803,Z 314.275,A -85,B 0,C 180,E1 -10873.899,E2 -10873.899} C_VEL
LIN {X 0,Y 406.228,Z 327.647,A -85,B 0,C 180,E1 -10874.704,E2 -10874.704} C_VEL
LIN {X 0,Y 405.568,Z 338.784,A -85,B 0,C 180,E1 -10875.577,E2 -10875.577} C_VEL
LIN {X 0,Y 404.894,Z 349.919,A -85,B 0,C 180,E1 -10876.677,E2 -10876.677} C_VEL
LIN {X 0,Y 404.265,Z 360.381,A -85,B 0,C 180,E1 -10877.96,E2 -10877.96} C_VEL
LIN {X 0,Y 403.774,Z 368.699,A -85,B 0,C 180,E1 -10879.217,E2 -10879.217} C_VEL
LIN {X 0,Y 403.419,Z 376.851,A -85,B 0,C 180,E1 -10880.728,E2 -10880.728} C_VEL
LIN {X 0,Y 403.215,Z 382.367,A -85,B 0,C 180,E1 -10881.986,E2 -10881.986} C_VEL
LIN {X 0,Y 403.056,Z 388.277,A -85,B 0,C 180,E1 -10883.668,E2 -10883.668} C_VEL
LIN {X 0,Y 403.103,Z 391.859,A -85,B 0,C 180,E1 -10885,E2 -10885} C_VEL
LIN {X 0,Y 403.023,Z 393.964,A -85,B 0,C 180,E1 -10886.002,E2 -10886.002} C_VEL
LIN {X 0,Y 403.132,Z 395.612,A -85,B 0,C 180,E1 -10887.003,E2 -10887.003} C_VEL
LIN {X 0,Y 403.091,Z 396.822,A -85,B 0,C 180,E1 -10888.003,E2 -10888.003} C_VEL
LIN {X 0,Y 403.125,Z 397.581,A -85,B 0,C 180,E1 -10889.002,E2 -10889.002} C_VEL
LIN {X 0,Y 403.16,Z 397.892,A -85,B 0,C 180,E1 -10890.001,E2 -10890.001} C_VEL
LIN {X 0,Y 403.099,Z 397.783,A -85,B 0,C 180,E1 -10891,E2 -10891} C_VEL
LIN {X 0,Y 403.086,Z 397.256,A -85,B 0,C 180,E1 -10892,E2 -10892} C_VEL
LIN {X 0,Y 403.085,Z 396.258,A -85,B 0,C 180,E1 -10893,E2 -10893} C_VEL
LIN {X 0,Y 403.02,Z 394.838,A -85,B 0,C 180,E1 -10894.001,E2 -10894.001} C_VEL
LIN {X 0,Y 403.045,Z 391.875,A -85,B 0,C 180,E1 -10895.505,E2 -10895.505} C_VEL
LIN {X 0,Y 403.108,Z 387.838,A -85,B 0,C 180,E1 -10897.011,E2 -10897.011} C_VEL
LIN {X 0,Y 403.382,Z 381.666,A -85,B 0,C 180,E1 -10898.77,E2 -10898.77} C_VEL
LIN {X 0,Y 403.769,Z 374.9,A -85,B 0,C 180,E1 -10900.278,E2 -10900.278} C_VEL
LIN {X 0,Y 404.409,Z 366.579,A -85,B 0,C 180,E1 -10901.784,E2 -10901.784} C_VEL
LIN {X 0,Y 405.151,Z 356.917,A -85,B 0,C 180,E1 -10903.207,E2 -10903.207} C_VEL
LIN {X 0,Y 405.942,Z 346.874,A -85,B 0,C 180,E1 -10904.412,E2 -10904.412} C_VEL
LIN {X 0,Y 407.019,Z 335.491,A -85,B 0,C 180,E1 -10905.525,E2 -10905.525} C_VEL
LIN {X 0,Y 408.088,Z 322.691,A -85,B 0,C 180,E1 -10906.51,E2 -10906.51} C_VEL
LIN {X 0,Y 408.457,Z 312.785,A -85,B 0,C 180,E1 -10907.14,E2 -10907.14} C_VEL
LIN {X 0,Y 408.076,Z 299.864,A -85,B 0,C 180,E1 -10907.831,E2 -10907.831} C_VEL
LIN {X 0,Y 406.235,Z 284.318,A -85,B 0,C 180,E1 -10908.515,E2 -10908.515} C_VEL
LIN {X 0,Y 404.886,Z 276.289,A -85,B 0,C 180,E1 -10908.896,E2 -10908.896} C_VEL
LIN {X 0,Y 404.777,Z 273.986,A -85,B 0,C 180,E1 -10909.118,E2 -10909.118} C_VEL
LIN {X 0,Y 406.164,Z 256.998,A -85,B 0,C 180,E1 -10912.914,E2 -10912.914} C_VEL
LIN {X 0,Y 407.774,Z 240.227,A -85,B 0,C 180,E1 -10916.624,E2 -10916.624} C_VEL
LIN {X 0,Y 409.814,Z 223.444,A -85,B 0,C 180,E1 -10920.392,E2 -10920.392} C_VEL
LIN {X 0,Y 410.139,Z 220.64,A -85,B 0,C 180,E1 -10921.043,E2 -10921.043} C_VEL
LIN {X 0,Y 409.44,Z 216.273,A -85,B 0,C 180,E1 -10922.149,E2 -10922.149} C_VEL
LIN {X 0,Y 407.009,Z 205.143,A -85,B 0,C 180,E1 -10925.184,E2 -10925.184} C_VEL
LIN {X 0,Y 404.166,Z 193.142,A -85,B 0,C 180,E1 -10928.797,E2 -10928.797} C_VEL
LIN {X 0,Y 404.128,Z 193.145,A -85,B 0,C 180,E1 -10931.6,E2 -10931.6} C_VEL
LIN {X 0,Y 404.15,Z 193.145,A -85,B 0,C 180,E1 -10934.523,E2 -10934.523} C_VEL
LIN {X 0,Y 404.132,Z 193.191,A -85,B 0,C 180,E1 -10936.194,E2 -10936.194} C_VEL
LIN {X 0,Y 405.374,Z 197.354,A -85,B 0,C 180,E1 -10938.791,E2 -10938.791} C_VEL
LIN {X 0,Y 406.916,Z 203.812,A -85,B 0,C 180,E1 -10942.173,E2 -10942.173} C_VEL
LIN {X 0,Y 407.667,Z 207.924,A -85,B 0,C 180,E1 -10944.123,E2 -10944.123} C_VEL
LIN {X 0,Y 407.552,Z 212.046,A -85,B 0,C 180,E1 -10945.868,E2 -10945.868} C_VEL
LIN {X 0,Y 406.609,Z 222.003,A -85,B 0,C 180,E1 -10949.917,E2 -10949.917} C_VEL
LIN {X 0,Y 406.168,Z 230.38,A -85,B 0,C 180,E1 -10953.264,E2 -10953.264} C_VEL
LIN {X 0,Y 405.776,Z 238.754,A -85,B 0,C 180,E1 -10956.631,E2 -10956.631} C_VEL
LIN {X 0,Y 405.334,Z 247.728,A -85,B 0,C 180,E1 -10960.238,E2 -10960.238} C_VEL
LIN {X 0,Y 405.248,Z 250.346,A -85,B 0,C 180,E1 -10961.287,E2 -10961.287} C_VEL
LIN {X 0,Y 408.932,Z 262.768,A -85,B 0,C 180,E1 -10962.079,E2 -10962.079} C_VEL
LIN {X 0,Y 410.417,Z 269.857,A -85,B 0,C 180,E1 -10962.56,E2 -10962.56} C_VEL
LIN {X 0,Y 409.711,Z 281.971,A -85,B 0,C 180,E1 -10963.302,E2 -10963.302} C_VEL
LIN {X 0,Y 408.773,Z 293.971,A -85,B 0,C 180,E1 -10964.248,E2 -10964.248} C_VEL
LIN {X 0,Y 407.769,Z 305.616,A -85,B 0,C 180,E1 -10965.4,E2 -10965.4} C_VEL
LIN {X 0,Y 406.849,Z 314.758,A -85,B 0,C 180,E1 -10966.514,E2 -10966.514} C_VEL
LIN {X 0,Y 405.975,Z 323.189,A -85,B 0,C 180,E1 -10967.757,E2 -10967.757} C_VEL
LIN {X 0,Y 405.211,Z 331.508,A -85,B 0,C 180,E1 -10969.254,E2 -10969.254} C_VEL
LIN {X 0,Y 404.673,Z 337.179,A -85,B 0,C 180,E1 -10970.504,E2 -10970.504} C_VEL
LIN {X 0,Y 404.116,Z 342.773,A -85,B 0,C 180,E1 -10972.003,E2 -10972.003} C_VEL
LIN {X 0,Y 403.667,Z 347.156,A -85,B 0,C 180,E1 -10973.502,E2 -10973.502} C_VEL
LIN {X 0,Y 403.523,Z 350.429,A -85,B 0,C 180,E1 -10975.004,E2 -10975.004} C_VEL
LIN {X 0,Y 403.371,Z 352.043,A -85,B 0,C 180,E1 -10976.004,E2 -10976.004} C_VEL
LIN {X 0,Y 403.21,Z 353.254,A -85,B 0,C 180,E1 -10977.003,E2 -10977.003} C_VEL
LIN {X 0,Y 403.09,Z 354.068,A -85,B 0,C 180,E1 -10978.002,E2 -10978.002} C_VEL
LIN {X 0,Y 402.999,Z 354.438,A -85,B 0,C 180,E1 -10979.001,E2 -10979.001} C_VEL
LIN {X 0,Y 402.951,Z 354.392,A -85,B 0,C 180,E1 -10980,E2 -10980} C_VEL
LIN {X 0,Y 402.958,Z 353.95,A -85,B 0,C 180,E1 -10980.999,E2 -10980.999} C_VEL
LIN {X 0,Y 403.022,Z 353.095,A -85,B 0,C 180,E1 -10981.999,E2 -10981.999} C_VEL
LIN {X 0,Y 403.152,Z 351.786,A -85,B 0,C 180,E1 -10982.998,E2 -10982.998} C_VEL
LIN {X 0,Y 403.13,Z 349.046,A -85,B 0,C 180,E1 -10984.5,E2 -10984.5} C_VEL
LIN {X 0,Y 403.337,Z 345.256,A -85,B 0,C 180,E1 -10986.001,E2 -10986.001} C_VEL
LIN {X 0,Y 403.563,Z 340.323,A -85,B 0,C 180,E1 -10987.505,E2 -10987.505} C_VEL
LIN {X 0,Y 403.944,Z 334.112,A -85,B 0,C 180,E1 -10989.009,E2 -10989.009} C_VEL
LIN {X 0,Y 404.401,Z 326.383,A -85,B 0,C 180,E1 -10990.514,E2 -10990.514} C_VEL
LIN {X 0,Y 405.05,Z 316.744,A -85,B 0,C 180,E1 -10992.018,E2 -10992.018} C_VEL
LIN {X 0,Y 405.732,Z 306.854,A -85,B 0,C 180,E1 -10993.269,E2 -10993.269} C_VEL
LIN {X 0,Y 406.337,Z 295.831,A -85,B 0,C 180,E1 -10994.399,E2 -10994.399} C_VEL
LIN {X 0,Y 407.011,Z 283.636,A -85,B 0,C 180,E1 -10995.396,E2 -10995.396} C_VEL
LIN {X 0,Y 407.717,Z 270.422,A -85,B 0,C 180,E1 -10996.219,E2 -10996.219} C_VEL
LIN {X 0,Y 407.635,Z 266.411,A -85,B 0,C 180,E1 -10996.432,E2 -10996.432} C_VEL
LIN {X 0,Y 405.205,Z 252.923,A -85,B 0,C 180,E1 -10997.08,E2 -10997.08} C_VEL
LIN {X 0,Y 404.062,Z 246.77,A -85,B 0,C 180,E1 -10997.316,E2 -10997.316} C_VEL
LIN {X 0,Y 404.271,Z 237.642,A -85,B 0,C 180,E1 -11000.878,E2 -11000.878} C_VEL
LIN {X 0,Y 404.499,Z 229.428,A -85,B 0,C 180,E1 -11004.098,E2 -11004.098} C_VEL
LIN {X 0,Y 404.739,Z 220.357,A -85,B 0,C 180,E1 -11007.675,E2 -11007.675} C_VEL
LIN {X 0,Y 405.052,Z 212.511,A -85,B 0,C 180,E1 -11010.787,E2 -11010.787} C_VEL
LIN {X 0,Y 405.254,Z 203.593,A -85,B 0,C 180,E1 -11014.307,E2 -11014.307} C_VEL
LIN {X 0,Y 405.141,Z 198.962,A -85,B 0,C 180,E1 -11016.143,E2 -11016.143} C_VEL
LIN {X 0,Y 404.228,Z 193.134,A -85,B 0,C 180,E1 -11018.589,E2 -11018.589} C_VEL
LIN {X 0,Y 404.124,Z 193.147,A -85,B 0,C 180,E1 -11021.599,E2 -11021.599} C_VEL
LIN {X 0,Y 404.15,Z 193.142,A -85,B 0,C 180,E1 -11024.521,E2 -11024.521} C_VEL
LIN {X 0,Y 404.142,Z 193.144,A -85,B 0,C 180,E1 -11027.295,E2 -11027.295} C_VEL
LIN {X 0,Y 404.14,Z 193.144,A -85,B 0,C 180,E1 -11029.951,E2 -11029.951} C_VEL
LIN {X 0,Y 404.137,Z 193.147,A -85,B 0,C 180,E1 -11033.125,E2 -11033.125} C_VEL
LIN {X 0,Y 404.143,Z 193.145,A -85,B 0,C 180,E1 -11036.186,E2 -11036.186} C_VEL
LIN {X 0,Y 404.124,Z 193.148,A -85,B 0,C 180,E1 -11038.551,E2 -11038.551} C_VEL
LIN {X 0,Y 404.003,Z 193.188,A -85,B 0,C 180,E1 -11040.85,E2 -11040.85} C_VEL
LIN {X 0,Y 403.962,Z 197.157,A -85,B 0,C 180,E1 -11044.217,E2 -11044.217} C_VEL
LIN {X 0,Y 403.892,Z 201.125,A -85,B 0,C 180,E1 -11047.491,E2 -11047.491} C_VEL
LIN {X 0,Y 403.777,Z 205.13,A -85,B 0,C 180,E1 -11050.687,E2 -11050.687} C_VEL
LIN {X 0,Y 403.769,Z 209.275,A -85,B 0,C 180,E1 -11053.828,E2 -11053.828} C_VEL
LIN {X 0,Y 403.799,Z 213.859,A -85,B 0,C 180,E1 -11057.076,E2 -11057.076} C_VEL
LIN {X 0,Y 403.817,Z 215.982,A -85,B 0,C 180,E1 -11058.485,E2 -11058.485} C_VEL
LIN {X 0,Y 406.445,Z 227.721,A -85,B 0,C 180,E1 -11059.097,E2 -11059.097} C_VEL
LIN {X 0,Y 407.085,Z 230.844,A -85,B 0,C 180,E1 -11059.304,E2 -11059.304} C_VEL
LIN {X 0,Y 406.919,Z 240.948,A -85,B 0,C 180,E1 -11060.053,E2 -11060.053} C_VEL
LIN {X 0,Y 406.541,Z 248.781,A -85,B 0,C 180,E1 -11060.85,E2 -11060.85} C_VEL
LIN {X 0,Y 406.229,Z 254.213,A -85,B 0,C 180,E1 -11061.542,E2 -11061.542} C_VEL
LIN {X 0,Y 405.846,Z 260.443,A -85,B 0,C 180,E1 -11062.536,E2 -11062.536} C_VEL
LIN {X 0,Y 405.353,Z 266.309,A -85,B 0,C 180,E1 -11063.778,E2 -11063.778} C_VEL
LIN {X 0,Y 405.07,Z 270.629,A -85,B 0,C 180,E1 -11065.022,E2 -11065.022} C_VEL
LIN {X 0,Y 404.807,Z 273.211,A -85,B 0,C 180,E1 -11066.017,E2 -11066.017} C_VEL
LIN {X 0,Y 404.445,Z 275.143,A -85,B 0,C 180,E1 -11067.011,E2 -11067.011} C_VEL
LIN {X 0,Y 404.399,Z 276.443,A -85,B 0,C 180,E1 -11068.007,E2 -11068.007} C_VEL
LIN {X 0,Y 404.277,Z 277.219,A -85,B 0,C 180,E1 -11069.003,E2 -11069.003} C_VEL
LIN {X 0,Y 404.226,Z 277.486,A -85,B 0,C 180,E1 -11069.999,E2 -11069.999} C_VEL
LIN {X 0,Y 404.271,Z 277.262,A -85,B 0,C 180,E1 -11070.995,E2 -11070.995} C_VEL
LIN {X 0,Y 404.382,Z 276.54,A -85,B 0,C 180,E1 -11071.991,E2 -11071.991} C_VEL
LIN {X 0,Y 404.44,Z 275.297,A -85,B 0,C 180,E1 -11072.987,E2 -11072.987} C_VEL
LIN {X 0,Y 404.99,Z 272.252,A -85,B 0,C 180,E1 -11074.478,E2 -11074.478} C_VEL
LIN {X 0,Y 405.124,Z 267.717,A -85,B 0,C 180,E1 -11075.962,E2 -11075.962} C_VEL
LIN {X 0,Y 404.57,Z 265.962,A -85,B 0,C 180,E1 -11076.467,E2 -11076.467} C_VEL
LIN {X 0,Y 402.049,Z 263.017,A -85,B 0,C 180,E1 -11077.259,E2 -11077.259} C_VEL
LIN {X 0,Y 399.616,Z 259.576,A -85,B 0,C 180,E1 -11078.01,E2 -11078.01} C_VEL
LIN {X 0,Y 399.191,Z 257.001,A -85,B 0,C 180,E1 -11078.444,E2 -11078.444} C_VEL
LIN {X 0,Y 399.622,Z 250.889,A -85,B 0,C 180,E1 -11079.286,E2 -11079.286} C_VEL
LIN {X 0,Y 399.949,Z 243.234,A -85,B 0,C 180,E1 -11080.119,E2 -11080.119} C_VEL
LIN {X 0,Y 400.297,Z 235.62,A -85,B 0,C 180,E1 -11080.749,E2 -11080.749} C_VEL
LIN {X 0,Y 399.983,Z 230.868,A -85,B 0,C 180,E1 -11081.079,E2 -11081.079} C_VEL
LIN {X 0,Y 397.733,Z 220.685,A -85,B 0,C 180,E1 -11081.675,E2 -11081.675} C_VEL
LIN {X 0,Y 396.78,Z 216.6,A -85,B 0,C 180,E1 -11081.881,E2 -11081.881} C_VEL
LIN {X 0,Y 396.724,Z 211.497,A -85,B 0,C 180,E1 -11085.409,E2 -11085.409} C_VEL
LIN {X 0,Y 396.751,Z 208.617,A -85,B 0,C 180,E1 -11087.524,E2 -11087.524} C_VEL
LIN {X 0,Y 396.754,Z 204.468,A -85,B 0,C 180,E1 -11090.747,E2 -11090.747} C_VEL
LIN {X 0,Y 396.864,Z 200.455,A -85,B 0,C 180,E1 -11094.034,E2 -11094.034} C_VEL
LIN {X 0,Y 396.973,Z 196.414,A -85,B 0,C 180,E1 -11097.405,E2 -11097.405} C_VEL
LIN {X 0,Y 396.986,Z 194.037,A -85,B 0,C 180,E1 -11099.714,E2 -11099.714} C_VEL
LIN {X 0,Y 397.11,Z 194.021,A -85,B 0,C 180,E1 -11103.271,E2 -11103.271} C_VEL
LIN {X 0,Y 397.104,Z 194.022,A -85,B 0,C 180,E1 -11105.733,E2 -11105.733} C_VEL
LIN {X 0,Y 397.109,Z 194.02,A -85,B 0,C 180,E1 -11109.576,E2 -11109.576} C_VEL
LIN {X 0,Y 397.098,Z 194.019,A -85,B 0,C 180,E1 -11113.478,E2 -11113.478} C_VEL
LIN {X 0,Y 397.095,Z 194.02,A -85,B 0,C 180,E1 -11116.52,E2 -11116.52} C_VEL
LIN {X 0,Y 397.107,Z 194.018,A -85,B 0,C 180,E1 -11120.422,E2 -11120.422} C_VEL
LIN {X 0,Y 397.101,Z 194.02,A -85,B 0,C 180,E1 -11124.264,E2 -11124.264} C_VEL
LIN {X 0,Y 397.106,Z 194.017,A -85,B 0,C 180,E1 -11126.726,E2 -11126.726} C_VEL
LIN {X 0,Y 397.125,Z 194.013,A -85,B 0,C 180,E1 -11130.296,E2 -11130.296} C_VEL
LIN {X 0,Y 397.185,Z 194.01,A -85,B 0,C 180,E1 -11132.609,E2 -11132.609} C_VEL
LIN {X 0,Y 397.123,Z 194.014,A -85,B 0,C 180,E1 -11135.981,E2 -11135.981} C_VEL
LIN {X 0,Y 397.128,Z 194.011,A -85,B 0,C 180,E1 -11139.704,E2 -11139.704} C_VEL
LIN {X 0,Y 397.173,Z 194.009,A -85,B 0,C 180,E1 -11142.843,E2 -11142.843} C_VEL
LIN {X 0,Y 397.168,Z 194.007,A -85,B 0,C 180,E1 -11145.656,E2 -11145.656} C_VEL
LIN {X 0,Y 397.189,Z 194.006,A -85,B 0,C 180,E1 -11148.776,E2 -11148.776} C_VEL
LIN {X 0,Y 397.349,Z 193.987,A -85,B 0,C 180,E1 -11152.076,E2 -11152.076} C_VEL
LIN {X 0,Y 397.241,Z 193.996,A -85,B 0,C 180,E1 -11154.925,E2 -11154.925} C_VEL
LIN {X 0,Y 397.44,Z 193.975,A -85,B 0,C 180,E1 -11157.973,E2 -11157.973} C_VEL
LIN {X 0,Y 397.568,Z 193.951,A -85,B 0,C 180,E1 -11160,E2 -11160} C_VEL
LIN {X 0,Y 397.361,Z 193.987,A -85,B 0,C 180,E1 -11163.042,E2 -11163.042} C_VEL
LIN {X 0,Y 397.35,Z 193.989,A -85,B 0,C 180,E1 -11167.112,E2 -11167.112} C_VEL
LIN {X 0,Y 397.204,Z 194.003,A -85,B 0,C 180,E1 -11170.191,E2 -11170.191} C_VEL
LIN {X 0,Y 397.215,Z 193.998,A -85,B 0,C 180,E1 -11173.321,E2 -11173.321} C_VEL
LIN {X 0,Y 397.17,Z 194.006,A -85,B 0,C 180,E1 -11177.156,E2 -11177.156} C_VEL
LIN {X 0,Y 397.091,Z 194.021,A -85,B 0,C 180,E1 -11180.731,E2 -11180.731} C_VEL
LIN {X 0,Y 397.095,Z 194.024,A -85,B 0,C 180,E1 -11184.021,E2 -11184.021} C_VEL
LIN {X 0,Y 397.054,Z 194.029,A -85,B 0,C 180,E1 -11187.401,E2 -11187.401} C_VEL
LIN {X 0,Y 397.088,Z 194.024,A -85,B 0,C 180,E1 -11189.864,E2 -11189.864} C_VEL
LIN {X 0,Y 397.108,Z 194.018,A -85,B 0,C 180,E1 -11193.719,E2 -11193.719} C_VEL
LIN {X 0,Y 397.082,Z 194.023,A -85,B 0,C 180,E1 -11197.209,E2 -11197.209} C_VEL
LIN {X 0,Y 397.048,Z 194.017,A -85,B 0,C 180,E1 -11200.439,E2 -11200.439} C_VEL
LIN {X 0,Y 397.092,Z 194.02,A -85,B 0,C 180,E1 -11203.65,E2 -11203.65} C_VEL
LIN {X 0,Y 397.095,Z 194.024,A -85,B 0,C 180,E1 -11206.522,E2 -11206.522} C_VEL
LIN {X 0,Y 397.161,Z 194.006,A -85,B 0,C 180,E1 -11210.63,E2 -11210.63} C_VEL
LIN {X 0,Y 399.66,Z 204.651,A -85,B 0,C 180,E1 -11213.99,E2 -11213.99} C_VEL
LIN {X 0,Y 402.039,Z 215.429,A -85,B 0,C 180,E1 -11217.044,E2 -11217.044} C_VEL
LIN {X 0,Y 403.247,Z 221.485,A -85,B 0,C 180,E1 -11218.649,E2 -11218.649} C_VEL
LIN {X 0,Y 402.108,Z 231.128,A -85,B 0,C 180,E1 -11220.915,E2 -11220.915} C_VEL
LIN {X 0,Y 399.975,Z 249.266,A -85,B 0,C 180,E1 -11225.059,E2 -11225.059} C_VEL
LIN {X 0,Y 398.438,Z 265.969,A -85,B 0,C 180,E1 -11228.857,E2 -11228.857} C_VEL
LIN {X 0,Y 397.281,Z 281.348,A -85,B 0,C 180,E1 -11232.433,E2 -11232.433} C_VEL
LIN {X 0,Y 399.246,Z 302.635,A -85,B 0,C 180,E1 -11233.154,E2 -11233.154} C_VEL
LIN {X 0,Y 399.838,Z 315.792,A -85,B 0,C 180,E1 -11233.799,E2 -11233.799} C_VEL
LIN {X 0,Y 399.217,Z 327.892,A -85,B 0,C 180,E1 -11234.559,E2 -11234.559} C_VEL
LIN {X 0,Y 398.546,Z 338.857,A -85,B 0,C 180,E1 -11235.448,E2 -11235.448} C_VEL
LIN {X 0,Y 397.835,Z 349.91,A -85,B 0,C 180,E1 -11236.567,E2 -11236.567} C_VEL
LIN {X 0,Y 397.222,Z 359.363,A -85,B 0,C 180,E1 -11237.743,E2 -11237.743} C_VEL
LIN {X 0,Y 396.759,Z 367.8,A -85,B 0,C 180,E1 -11239.024,E2 -11239.024} C_VEL
LIN {X 0,Y 396.375,Z 376.035,A -85,B 0,C 180,E1 -11240.562,E2 -11240.562} C_VEL
LIN {X 0,Y 396.166,Z 381.63,A -85,B 0,C 180,E1 -11241.842,E2 -11241.842} C_VEL
LIN {X 0,Y 396.009,Z 387.062,A -85,B 0,C 180,E1 -11243.378,E2 -11243.378} C_VEL
LIN {X 0,Y 396.029,Z 391.257,A -85,B 0,C 180,E1 -11244.911,E2 -11244.911} C_VEL
LIN {X 0,Y 395.94,Z 393.421,A -85,B 0,C 180,E1 -11245.93,E2 -11245.93} C_VEL
LIN {X 0,Y 396.044,Z 395.096,A -85,B 0,C 180,E1 -11246.95,E2 -11246.95} C_VEL
LIN {X 0,Y 396.018,Z 396.332,A -85,B 0,C 180,E1 -11247.967,E2 -11247.967} C_VEL
LIN {X 0,Y 396.039,Z 397.138,A -85,B 0,C 180,E1 -11248.985,E2 -11248.985} C_VEL
LIN {X 0,Y 396.084,Z 397.473,A -85,B 0,C 180,E1 -11250.001,E2 -11250.001} C_VEL
LIN {X 0,Y 396.015,Z 397.387,A -85,B 0,C 180,E1 -11251.018,E2 -11251.018} C_VEL
LIN {X 0,Y 396.011,Z 396.89,A -85,B 0,C 180,E1 -11252.035,E2 -11252.035} C_VEL
LIN {X 0,Y 395.982,Z 395.933,A -85,B 0,C 180,E1 -11253.053,E2 -11253.053} C_VEL
LIN {X 0,Y 395.935,Z 394.533,A -85,B 0,C 180,E1 -11254.073,E2 -11254.073} C_VEL
LIN {X 0,Y 395.937,Z 391.618,A -85,B 0,C 180,E1 -11255.604,E2 -11255.604} C_VEL
LIN {X 0,Y 396.031,Z 387.642,A -85,B 0,C 180,E1 -11257.137,E2 -11257.137} C_VEL
LIN {X 0,Y 396.286,Z 382.501,A -85,B 0,C 180,E1 -11258.671,E2 -11258.671} C_VEL
LIN {X 0,Y 396.697,Z 376.091,A -85,B 0,C 180,E1 -11260.206,E2 -11260.206} C_VEL
LIN {X 0,Y 397.287,Z 368.169,A -85,B 0,C 180,E1 -11261.739,E2 -11261.739} C_VEL
LIN {X 0,Y 398.151,Z 358.401,A -85,B 0,C 180,E1 -11263.267,E2 -11263.267} C_VEL
LIN {X 0,Y 398.857,Z 349.539,A -85,B 0,C 180,E1 -11264.413,E2 -11264.413} C_VEL
LIN {X 0,Y 399.949,Z 338.881,A -85,B 0,C 180,E1 -11265.545,E2 -11265.545} C_VEL
LIN {X 0,Y 401.08,Z 327.214,A -85,B 0,C 180,E1 -11266.545,E2 -11266.545} C_VEL
LIN {X 0,Y 401.873,Z 315.284,A -85,B 0,C 180,E1 -11267.374,E2 -11267.374} C_VEL
LIN {X 0,Y 401.609,Z 301.792,A -85,B 0,C 180,E1 -11268.153,E2 -11268.153} C_VEL
LIN {X 0,Y 400.113,Z 287.211,A -85,B 0,C 180,E1 -11268.851,E2 -11268.851} C_VEL
LIN {X 0,Y 398.309,Z 276.338,A -85,B 0,C 180,E1 -11269.368,E2 -11269.368} C_VEL
LIN {X 0,Y 397.909,Z 271.721,A -85,B 0,C 180,E1 -11269.811,E2 -11269.811} C_VEL
LIN {X 0,Y 399.257,Z 256.34,A -85,B 0,C 180,E1 -11273.333,E2 -11273.333} C_VEL
LIN {X 0,Y 400.822,Z 241.206,A -85,B 0,C 180,E1 -11276.77,E2 -11276.77} C_VEL
LIN {X 0,Y 402.841,Z 225.431,A -85,B 0,C 180,E1 -11280.395,E2 -11280.395} C_VEL
LIN {X 0,Y 403.13,Z 220.692,A -85,B 0,C 180,E1 -11281.535,E2 -11281.535} C_VEL
LIN {X 0,Y 400.545,Z 208.488,A -85,B 0,C 180,E1 -11284.869,E2 -11284.869} C_VEL
LIN {X 0,Y 397.658,Z 196.394,A -85,B 0,C 180,E1 -11288.545,E2 -11288.545} C_VEL
LIN {X 0,Y 397.166,Z 194.015,A -85,B 0,C 180,E1 -11289.371,E2 -11289.371} C_VEL
LIN {X 0,Y 397.107,Z 194.021,A -85,B 0,C 180,E1 -11293.48,E2 -11293.48} C_VEL
LIN {X 0,Y 397.136,Z 194.111,A -85,B 0,C 180,E1 -11293.983,E2 -11293.983} C_VEL
LIN {X 0,Y 398.043,Z 197.147,A -85,B 0,C 180,E1 -11296.481,E2 -11296.481} C_VEL
LIN {X 0,Y 399.288,Z 201.584,A -85,B 0,C 180,E1 -11299.364,E2 -11299.364} C_VEL
LIN {X 0,Y 400.431,Z 206.721,A -85,B 0,C 180,E1 -11302.168,E2 -11302.168} C_VEL
LIN {X 0,Y 401.07,Z 210.874,A -85,B 0,C 180,E1 -11304.211,E2 -11304.211} C_VEL
LIN {X 0,Y 400.691,Z 216.071,A -85,B 0,C 180,E1 -11306.461,E2 -11306.461} C_VEL
LIN {X 0,Y 399.77,Z 225.798,A -85,B 0,C 180,E1 -11310.512,E2 -11310.512} C_VEL
LIN {X 0,Y 399.26,Z 234.071,A -85,B 0,C 180,E1 -11313.892,E2 -11313.892} C_VEL
LIN {X 0,Y 398.834,Z 242.101,A -85,B 0,C 180,E1 -11317.19,E2 -11317.19} C_VEL
LIN {X 0,Y 398.41,Z 250.921,A -85,B 0,C 180,E1 -11320.789,E2 -11320.789} C_VEL
LIN {X 0,Y 401.941,Z 262.207,A -85,B 0,C 180,E1 -11321.547,E2 -11321.547} C_VEL
LIN {X 0,Y 403.98,Z 271.55,A -85,B 0,C 180,E1 -11322.211,E2 -11322.211} C_VEL
LIN {X 0,Y 403.076,Z 284.103,A -85,B 0,C 180,E1 -11323.019,E2 -11323.019} C_VEL
LIN {X 0,Y 402.028,Z 296.434,A -85,B 0,C 180,E1 -11324.047,E2 -11324.047} C_VEL
LIN {X 0,Y 401.019,Z 307.019,A -85,B 0,C 180,E1 -11325.149,E2 -11325.149} C_VEL
LIN {X 0,Y 400.058,Z 315.966,A -85,B 0,C 180,E1 -11326.281,E2 -11326.281} C_VEL
LIN {X 0,Y 399.147,Z 324.259,A -85,B 0,C 180,E1 -11327.544,E2 -11327.544} C_VEL
LIN {X 0,Y 398.388,Z 331.186,A -85,B 0,C 180,E1 -11328.811,E2 -11328.811} C_VEL
LIN {X 0,Y 397.732,Z 338.024,A -85,B 0,C 180,E1 -11330.336,E2 -11330.336} C_VEL
LIN {X 0,Y 397.145,Z 343.524,A -85,B 0,C 180,E1 -11331.861,E2 -11331.861} C_VEL
LIN {X 0,Y 396.65,Z 347.818,A -85,B 0,C 180,E1 -11333.387,E2 -11333.387} C_VEL
LIN {X 0,Y 396.48,Z 351.022,A -85,B 0,C 180,E1 -11334.915,E2 -11334.915} C_VEL
LIN {X 0,Y 396.328,Z 352.597,A -85,B 0,C 180,E1 -11335.933,E2 -11335.933} C_VEL
LIN {X 0,Y 396.152,Z 353.775,A -85,B 0,C 180,E1 -11336.949,E2 -11336.949} C_VEL
LIN {X 0,Y 396.019,Z 354.546,A -85,B 0,C 180,E1 -11337.966,E2 -11337.966} C_VEL
LIN {X 0,Y 395.923,Z 354.865,A -85,B 0,C 180,E1 -11338.983,E2 -11338.983} C_VEL
LIN {X 0,Y 395.873,Z 354.786,A -85,B 0,C 180,E1 -11340,E2 -11340} C_VEL
LIN {X 0,Y 395.884,Z 354.311,A -85,B 0,C 180,E1 -11341.017,E2 -11341.017} C_VEL
LIN {X 0,Y 395.955,Z 353.396,A -85,B 0,C 180,E1 -11342.034,E2 -11342.034} C_VEL
LIN {X 0,Y 396.069,Z 352.051,A -85,B 0,C 180,E1 -11343.052,E2 -11343.052} C_VEL
LIN {X 0,Y 396.055,Z 349.242,A -85,B 0,C 180,E1 -11344.58,E2 -11344.58} C_VEL
LIN {X 0,Y 396.306,Z 344.437,A -85,B 0,C 180,E1 -11346.434,E2 -11346.434} C_VEL
LIN {X 0,Y 396.61,Z 338.416,A -85,B 0,C 180,E1 -11348.15,E2 -11348.15} C_VEL
LIN {X 0,Y 397.089,Z 331.629,A -85,B 0,C 180,E1 -11349.68,E2 -11349.68} C_VEL
LIN {X 0,Y 397.602,Z 323.209,A -85,B 0,C 180,E1 -11351.212,E2 -11351.212} C_VEL
LIN {X 0,Y 398.241,Z 314.597,A -85,B 0,C 180,E1 -11352.485,E2 -11352.485} C_VEL
LIN {X 0,Y 398.899,Z 304.136,A -85,B 0,C 180,E1 -11353.76,E2 -11353.76} C_VEL
LIN {X 0,Y 399.542,Z 292.629,A -85,B 0,C 180,E1 -11354.886,E2 -11354.886} C_VEL
LIN {X 0,Y 400.202,Z 280.918,A -85,B 0,C 180,E1 -11355.795,E2 -11355.795} C_VEL
LIN {X 0,Y 400.791,Z 268.098,A -85,B 0,C 180,E1 -11356.563,E2 -11356.563} C_VEL
LIN {X 0,Y 398.322,Z 253.911,A -85,B 0,C 180,E1 -11357.274,E2 -11357.274} C_VEL
LIN {X 0,Y 397.015,Z 247.078,A -85,B 0,C 180,E1 -11357.547,E2 -11357.547} C_VEL
LIN {X 0,Y 397.27,Z 237.618,A -85,B 0,C 180,E1 -11361.264,E2 -11361.264} C_VEL
LIN {X 0,Y 397.467,Z 230.7,A -85,B 0,C 180,E1 -11363.997,E2 -11363.997} C_VEL
LIN {X 0,Y 397.69,Z 222.262,A -85,B 0,C 180,E1 -11367.353,E2 -11367.353} C_VEL
LIN {X 0,Y 398.031,Z 213.601,A -85,B 0,C 180,E1 -11370.801,E2 -11370.801} C_VEL
LIN {X 0,Y 398.236,Z 205.652,A -85,B 0,C 180,E1 -11373.956,E2 -11373.956} C_VEL
LIN {X 0,Y 398.128,Z 199.946,A -85,B 0,C 180,E1 -11376.254,E2 -11376.254} C_VEL
LIN {X 0,Y 397.179,Z 194.012,A -85,B 0,C 180,E1 -11378.781,E2 -11378.781} C_VEL
LIN {X 0,Y 397.07,Z 194.026,A -85,B 0,C 180,E1 -11382.267,E2 -11382.267} C_VEL
LIN {X 0,Y 397.092,Z 194.019,A -85,B 0,C 180,E1 -11385.068,E2 -11385.068} C_VEL
LIN {X 0,Y 397.071,Z 194.025,A -85,B 0,C 180,E1 -11388.021,E2 -11388.021} C_VEL
LIN {X 0,Y 397.107,Z 194.022,A -85,B 0,C 180,E1 -11391.143,E2 -11391.143} C_VEL
LIN {X 0,Y 397.103,Z 194.023,A -85,B 0,C 180,E1 -11394.501,E2 -11394.501} C_VEL
LIN {X 0,Y 397.071,Z 194.025,A -85,B 0,C 180,E1 -11397.927,E2 -11397.927} C_VEL
LIN {X 0,Y 396.992,Z 194.037,A -85,B 0,C 180,E1 -11400.284,E2 -11400.284} C_VEL
LIN {X 0,Y 396.959,Z 195.915,A -85,B 0,C 180,E1 -11402.28,E2 -11402.28} C_VEL
LIN {X 0,Y 396.933,Z 198.951,A -85,B 0,C 180,E1 -11404.852,E2 -11404.852} C_VEL
LIN {X 0,Y 396.812,Z 202.999,A -85,B 0,C 180,E1 -11408.164,E2 -11408.164} C_VEL
LIN {X 0,Y 396.72,Z 207.07,A -85,B 0,C 180,E1 -11411.404,E2 -11411.404} C_VEL
LIN {X 0,Y 396.746,Z 209.88,A -85,B 0,C 180,E1 -11413.534,E2 -11413.534} C_VEL
LIN {X 0,Y 396.774,Z 214.709,A -85,B 0,C 180,E1 -11416.96,E2 -11416.96} C_VEL
LIN {X 0,Y 396.805,Z 216.632,A -85,B 0,C 180,E1 -11418.246,E2 -11418.246} C_VEL
LIN {X 0,Y 399.159,Z 226.955,A -85,B 0,C 180,E1 -11418.767,E2 -11418.767} C_VEL
LIN {X 0,Y 400.247,Z 232.276,A -85,B 0,C 180,E1 -11419.119,E2 -11419.119} C_VEL
LIN {X 0,Y 400.03,Z 242.188,A -85,B 0,C 180,E1 -11419.88,E2 -11419.88} C_VEL
LIN {X 0,Y 399.643,Z 249.87,A -85,B 0,C 180,E1 -11420.686,E2 -11420.686} C_VEL
LIN {X 0,Y 399.295,Z 255.293,A -85,B 0,C 180,E1 -11421.395,E2 -11421.395} C_VEL
LIN {X 0,Y 398.875,Z 261.494,A -85,B 0,C 180,E1 -11422.405,E2 -11422.405} C_VEL
LIN {X 0,Y 398.373,Z 267.326,A -85,B 0,C 180,E1 -11423.668,E2 -11423.668} C_VEL
LIN {X 0,Y 398.074,Z 271.622,A -85,B 0,C 180,E1 -11424.934,E2 -11424.934} C_VEL
LIN {X 0,Y 397.805,Z 274.195,A -85,B 0,C 180,E1 -11425.946,E2 -11425.946} C_VEL
LIN {X 0,Y 397.431,Z 276.121,A -85,B 0,C 180,E1 -11426.958,E2 -11426.958} C_VEL
LIN {X 0,Y 397.379,Z 277.418,A -85,B 0,C 180,E1 -11427.972,E2 -11427.972} C_VEL
LIN {X 0,Y 397.253,Z 278.193,A -85,B 0,C 180,E1 -11428.985,E2 -11428.985} C_VEL
LIN {X 0,Y 397.201,Z 278.46,A -85,B 0,C 180,E1 -11429.999,E2 -11429.999} C_VEL
LIN {X 0,Y 397.248,Z 278.235,A -85,B 0,C 180,E1 -11431.012,E2 -11431.012} C_VEL
LIN {X 0,Y 397.364,Z 277.514,A -85,B 0,C 180,E1 -11432.026,E2 -11432.026} C_VEL
LIN {X 0,Y 397.426,Z 276.274,A -85,B 0,C 180,E1 -11433.04,E2 -11433.04} C_VEL
LIN {X 0,Y 397.992,Z 273.238,A -85,B 0,C 180,E1 -11434.556,E2 -11434.556} C_VEL
LIN {X 0,Y 398.137,Z 268.683,A -85,B 0,C 180,E1 -11436.078,E2 -11436.078} C_VEL
LIN {X 0,Y 398.564,Z 265.648,A -85,B 0,C 180,E1 -11436.834,E2 -11436.834} C_VEL
LIN {X 0,Y 398.818,Z 261.957,A -85,B 0,C 180,E1 -11437.593,E2 -11437.593} C_VEL
LIN {X 0,Y 399.191,Z 257.001,A -85,B 0,C 180,E1 -11438.444,E2 -11438.444} C_VEL
LIN {X 0,Y 399.036,Z 252.968,A -85,B 0,C 180,E1 -11439.048,E2 -11439.048} C_VEL
LIN {X 0,Y 397.678,Z 247.217,A -85,B 0,C 180,E1 -11439.808,E2 -11439.808} C_VEL
LIN {X 0,Y 395.191,Z 239.596,A -85,B 0,C 180,E1 -11440.653,E2 -11440.653} C_VEL
LIN {X 0,Y 393.293,Z 232.95,A -85,B 0,C 180,E1 -11441.227,E2 -11441.227} C_VEL
LIN {X 0,Y 391.003,Z 222.434,A -85,B 0,C 180,E1 -11441.882,E2 -11441.882} C_VEL
LIN {X 0,Y 389.767,Z 217.249,A -85,B 0,C 180,E1 -11442.131,E2 -11442.131} C_VEL
LIN {X 0,Y 389.692,Z 212.136,A -85,B 0,C 180,E1 -11445.694,E2 -11445.694} C_VEL
LIN {X 0,Y 389.721,Z 207.784,A -85,B 0,C 180,E1 -11448.94,E2 -11448.94} C_VEL
LIN {X 0,Y 389.784,Z 203.651,A -85,B 0,C 180,E1 -11452.248,E2 -11452.248} C_VEL
LIN {X 0,Y 389.893,Z 199.525,A -85,B 0,C 180,E1 -11455.674,E2 -11455.674} C_VEL
LIN {X 0,Y 389.908,Z 195.478,A -85,B 0,C 180,E1 -11459.12,E2 -11459.12} C_VEL
LIN {X 0,Y 389.946,Z 194.913,A -85,B 0,C 180,E1 -11460.306,E2 -11460.306} C_VEL
LIN {X 0,Y 390.035,Z 194.9,A -85,B 0,C 180,E1 -11462.72,E2 -11462.72} C_VEL
LIN {X 0,Y 390.053,Z 194.899,A -85,B 0,C 180,E1 -11465.824,E2 -11465.824} C_VEL
LIN {X 0,Y 390.066,Z 194.899,A -85,B 0,C 180,E1 -11469.217,E2 -11469.217} C_VEL
LIN {X 0,Y 390.038,Z 194.898,A -85,B 0,C 180,E1 -11472.373,E2 -11472.373} C_VEL
LIN {X 0,Y 390.039,Z 194.9,A -85,B 0,C 180,E1 -11475.353,E2 -11475.353} C_VEL
LIN {X 0,Y 390.024,Z 194.901,A -85,B 0,C 180,E1 -11478.185,E2 -11478.185} C_VEL
LIN {X 0,Y 390.085,Z 194.896,A -85,B 0,C 180,E1 -11480.907,E2 -11480.907} C_VEL
LIN {X 0,Y 390.077,Z 194.896,A -85,B 0,C 180,E1 -11484.792,E2 -11484.792} C_VEL
LIN {X 0,Y 390.04,Z 194.902,A -85,B 0,C 180,E1 -11488.497,E2 -11488.497} C_VEL
LIN {X 0,Y 390.107,Z 194.891,A -85,B 0,C 180,E1 -11492.069,E2 -11492.069} C_VEL
LIN {X 0,Y 390.07,Z 194.888,A -85,B 0,C 180,E1 -11495.518,E2 -11495.518} C_VEL
LIN {X 0,Y 390.045,Z 194.893,A -85,B 0,C 180,E1 -11498.877,E2 -11498.877} C_VEL
LIN {X 0,Y 390.118,Z 194.89,A -85,B 0,C 180,E1 -11502.166,E2 -11502.166} C_VEL
LIN {X 0,Y 390.136,Z 194.88,A -85,B 0,C 180,E1 -11505.392,E2 -11505.392} C_VEL
LIN {X 0,Y 390.138,Z 194.884,A -85,B 0,C 180,E1 -11508.571,E2 -11508.571} C_VEL
LIN {X 0,Y 390.296,Z 194.865,A -85,B 0,C 180,E1 -11512.031,E2 -11512.031} C_VEL
LIN {X 0,Y 390.213,Z 194.872,A -85,B 0,C 180,E1 -11514.833,E2 -11514.833} C_VEL
LIN {X 0,Y 390.409,Z 194.851,A -85,B 0,C 180,E1 -11517.937,E2 -11517.937} C_VEL
LIN {X 0,Y 390.538,Z 194.827,A -85,B 0,C 180,E1 -11520,E2 -11520} C_VEL
LIN {X 0,Y 390.295,Z 194.866,A -85,B 0,C 180,E1 -11523.097,E2 -11523.097} C_VEL
LIN {X 0,Y 390.315,Z 194.862,A -85,B 0,C 180,E1 -11526.202,E2 -11526.202} C_VEL
LIN {X 0,Y 390.303,Z 194.867,A -85,B 0,C 180,E1 -11528.282,E2 -11528.282} C_VEL
LIN {X 0,Y 390.158,Z 194.883,A -85,B 0,C 180,E1 -11532.483,E2 -11532.483} C_VEL
LIN {X 0,Y 390.127,Z 194.889,A -85,B 0,C 180,E1 -11535.677,E2 -11535.677} C_VEL
LIN {X 0,Y 390.09,Z 194.893,A -85,B 0,C 180,E1 -11538.923,E2 -11538.923} C_VEL
LIN {X 0,Y 390.023,Z 194.904,A -85,B 0,C 180,E1 -11542.235,E2 -11542.235} C_VEL
LIN {X 0,Y 390.039,Z 194.903,A -85,B 0,C 180,E1 -11545.723,E2 -11545.723} C_VEL
LIN {X 0,Y 390.013,Z 194.904,A -85,B 0,C 180,E1 -11549.113,E2 -11549.113} C_VEL
LIN {X 0,Y 390.033,Z 194.899,A -85,B 0,C 180,E1 -11552.723,E2 -11552.723} C_VEL
LIN {X 0,Y 390.045,Z 194.901,A -85,B 0,C 180,E1 -11555.826,E2 -11555.826} C_VEL
LIN {X 0,Y 390.029,Z 194.901,A -85,B 0,C 180,E1 -11559.214,E2 -11559.214} C_VEL
LIN {X 0,Y 390.028,Z 194.902,A -85,B 0,C 180,E1 -11562.374,E2 -11562.374} C_VEL
LIN {X 0,Y 390.037,Z 194.9,A -85,B 0,C 180,E1 -11565.356,E2 -11565.356} C_VEL
LIN {X 0,Y 390.024,Z 194.892,A -85,B 0,C 180,E1 -11568.188,E2 -11568.188} C_VEL
LIN {X 0,Y 390.125,Z 195.093,A -85,B 0,C 180,E1 -11570.214,E2 -11570.214} C_VEL
LIN {X 0,Y 392.816,Z 206.376,A -85,B 0,C 180,E1 -11573.816,E2 -11573.816} C_VEL
LIN {X 0,Y 395.032,Z 216.431,A -85,B 0,C 180,E1 -11576.739,E2 -11576.739} C_VEL
LIN {X 0,Y 396.274,Z 222.338,A -85,B 0,C 180,E1 -11578.352,E2 -11578.352} C_VEL
LIN {X 0,Y 396.032,Z 226.264,A -85,B 0,C 180,E1 -11579.325,E2 -11579.325} C_VEL
LIN {X 0,Y 393.856,Z 242.46,A -85,B 0,C 180,E1 -11583.152,E2 -11583.152} C_VEL
LIN {X 0,Y 392.181,Z 258.072,A -85,B 0,C 180,E1 -11586.783,E2 -11586.783} C_VEL
LIN {X 0,Y 390.754,Z 274.115,A -85,B 0,C 180,E1 -11590.567,E2 -11590.567} C_VEL
LIN {X 0,Y 390.26,Z 280.926,A -85,B 0,C 180,E1 -11592.204,E2 -11592.204} C_VEL
LIN {X 0,Y 392.132,Z 301.418,A -85,B 0,C 180,E1 -11592.897,E2 -11592.897} C_VEL
LIN {X 0,Y 392.782,Z 313.792,A -85,B 0,C 180,E1 -11593.5,E2 -11593.5} C_VEL
LIN {X 0,Y 392.431,Z 324.394,A -85,B 0,C 180,E1 -11594.152,E2 -11594.152} C_VEL
LIN {X 0,Y 391.677,Z 336.004,A -85,B 0,C 180,E1 -11595.054,E2 -11595.054} C_VEL
LIN {X 0,Y 391.097,Z 344.929,A -85,B 0,C 180,E1 -11595.912,E2 -11595.912} C_VEL
LIN {X 0,Y 390.552,Z 354.365,A -85,B 0,C 180,E1 -11597.002,E2 -11597.002} C_VEL
LIN {X 0,Y 389.946,Z 363.625,A -85,B 0,C 180,E1 -11598.303,E2 -11598.303} C_VEL
LIN {X 0,Y 389.382,Z 372.604,A -85,B 0,C 180,E1 -11599.866,E2 -11599.866} C_VEL
LIN {X 0,Y 389.126,Z 379.839,A -85,B 0,C 180,E1 -11601.432,E2 -11601.432} C_VEL
LIN {X 0,Y 388.963,Z 384.693,A -85,B 0,C 180,E1 -11602.735,E2 -11602.735} C_VEL
LIN {X 0,Y 388.865,Z 388.701,A -85,B 0,C 180,E1 -11604.058,E2 -11604.058} C_VEL
LIN {X 0,Y 388.912,Z 391.793,A -85,B 0,C 180,E1 -11605.337,E2 -11605.337} C_VEL
LIN {X 0,Y 388.959,Z 394.562,A -85,B 0,C 180,E1 -11606.894,E2 -11606.894} C_VEL
LIN {X 0,Y 388.947,Z 395.827,A -85,B 0,C 180,E1 -11607.93,E2 -11607.93} C_VEL
LIN {X 0,Y 388.957,Z 396.673,A -85,B 0,C 180,E1 -11608.966,E2 -11608.966} C_VEL
LIN {X 0,Y 388.998,Z 397.052,A -85,B 0,C 180,E1 -11610.001,E2 -11610.001} C_VEL
LIN {X 0,Y 388.935,Z 396.99,A -85,B 0,C 180,E1 -11611.037,E2 -11611.037} C_VEL
LIN {X 0,Y 388.938,Z 396.519,A -85,B 0,C 180,E1 -11612.072,E2 -11612.072} C_VEL
LIN {X 0,Y 388.88,Z 395.614,A -85,B 0,C 180,E1 -11613.109,E2 -11613.109} C_VEL
LIN {X 0,Y 388.852,Z 394.244,A -85,B 0,C 180,E1 -11614.147,E2 -11614.147} C_VEL
LIN {X 0,Y 388.83,Z 390.945,A -85,B 0,C 180,E1 -11615.903,E2 -11615.903} C_VEL
LIN {X 0,Y 389.048,Z 385.939,A -85,B 0,C 180,E1 -11617.788,E2 -11617.788} C_VEL
LIN {X 0,Y 389.418,Z 379.404,A -85,B 0,C 180,E1 -11619.611,E2 -11619.611} C_VEL
LIN {X 0,Y 389.902,Z 372.386,A -85,B 0,C 180,E1 -11621.174,E2 -11621.174} C_VEL
LIN {X 0,Y 390.813,Z 363.73,A -85,B 0,C 180,E1 -11622.727,E2 -11622.727} C_VEL
LIN {X 0,Y 391.58,Z 353.905,A -85,B 0,C 180,E1 -11624.176,E2 -11624.176} C_VEL
LIN {X 0,Y 392.779,Z 343.303,A -85,B 0,C 180,E1 -11625.437,E2 -11625.437} C_VEL
LIN {X 0,Y 394.036,Z 331.37,A -85,B 0,C 180,E1 -11626.582,E2 -11626.582} C_VEL
LIN {X 0,Y 395.122,Z 319.889,A -85,B 0,C 180,E1 -11627.468,E2 -11627.468} C_VEL
LIN {X 0,Y 395.302,Z 306.505,A -85,B 0,C 180,E1 -11628.328,E2 -11628.328} C_VEL
LIN {X 0,Y 394.288,Z 292.629,A -85,B 0,C 180,E1 -11629.08,E2 -11629.08} C_VEL
LIN {X 0,Y 391.913,Z 277.565,A -85,B 0,C 180,E1 -11629.822,E2 -11629.822} C_VEL
LIN {X 0,Y 391.555,Z 275.756,A -85,B 0,C 180,E1 -11629.941,E2 -11629.941} C_VEL
LIN {X 0,Y 391.102,Z 269.374,A -85,B 0,C 180,E1 -11630.554,E2 -11630.554} C_VEL
LIN {X 0,Y 392.51,Z 254.452,A -85,B 0,C 180,E1 -11634.053,E2 -11634.053} C_VEL
LIN {X 0,Y 394.25,Z 239.169,A -85,B 0,C 180,E1 -11637.613,E2 -11637.613} C_VEL
LIN {X 0,Y 396.205,Z 225.019,A -85,B 0,C 180,E1 -11640.959,E2 -11640.959} C_VEL
LIN {X 0,Y 396.254,Z 222.266,A -85,B 0,C 180,E1 -11641.643,E2 -11641.643} C_VEL
LIN {X 0,Y 393.569,Z 209.71,A -85,B 0,C 180,E1 -11645.163,E2 -11645.163} C_VEL
LIN {X 0,Y 390.87,Z 198.357,A -85,B 0,C 180,E1 -11648.678,E2 -11648.678} C_VEL
LIN {X 0,Y 390.222,Z 195.608,A -85,B 0,C 180,E1 -11649.616,E2 -11649.616} C_VEL
LIN {X 0,Y 390.567,Z 196.821,A -85,B 0,C 180,E1 -11652.458,E2 -11652.458} C_VEL
LIN {X 0,Y 391.214,Z 198.457,A -85,B 0,C 180,E1 -11654.478,E2 -11654.478} C_VEL
LIN {X 0,Y 392.168,Z 201.768,A -85,B 0,C 180,E1 -11657.288,E2 -11657.288} C_VEL
LIN {X 0,Y 393.268,Z 206.255,A -85,B 0,C 180,E1 -11660.216,E2 -11660.216} C_VEL
LIN {X 0,Y 394.13,Z 210.663,A -85,B 0,C 180,E1 -11662.679,E2 -11662.679} C_VEL
LIN {X 0,Y 394.473,Z 214.507,A -85,B 0,C 180,E1 -11664.618,E2 -11664.618} C_VEL
LIN {X 0,Y 393.82,Z 219.963,A -85,B 0,C 180,E1 -11667.01,E2 -11667.01} C_VEL
LIN {X 0,Y 393.058,Z 228.337,A -85,B 0,C 180,E1 -11670.547,E2 -11670.547} C_VEL
LIN {X 0,Y 392.442,Z 236.631,A -85,B 0,C 180,E1 -11674.04,E2 -11674.04} C_VEL
LIN {X 0,Y 391.983,Z 244.48,A -85,B 0,C 180,E1 -11677.326,E2 -11677.326} C_VEL
LIN {X 0,Y 391.627,Z 251.619,A -85,B 0,C 180,E1 -11680.252,E2 -11680.252} C_VEL
LIN {X 0,Y 395.518,Z 263.759,A -85,B 0,C 180,E1 -11681.123,E2 -11681.123} C_VEL
LIN {X 0,Y 397.549,Z 273.052,A -85,B 0,C 180,E1 -11681.827,E2 -11681.827} C_VEL
LIN {X 0,Y 396.483,Z 286.308,A -85,B 0,C 180,E1 -11682.728,E2 -11682.728} C_VEL
LIN {X 0,Y 395.496,Z 297.042,A -85,B 0,C 180,E1 -11683.658,E2 -11683.658} C_VEL
LIN {X 0,Y 394.302,Z 308.499,A -85,B 0,C 180,E1 -11684.89,E2 -11684.89} C_VEL
LIN {X 0,Y 393.277,Z 317.252,A -85,B 0,C 180,E1 -11686.04,E2 -11686.04} C_VEL
LIN {X 0,Y 392.312,Z 325.396,A -85,B 0,C 180,E1 -11687.323,E2 -11687.323} C_VEL
LIN {X 0,Y 391.507,Z 332.189,A -85,B 0,C 180,E1 -11688.611,E2 -11688.611} C_VEL
LIN {X 0,Y 390.797,Z 338.912,A -85,B 0,C 180,E1 -11690.163,E2 -11690.163} C_VEL
LIN {X 0,Y 390.16,Z 344.29,A -85,B 0,C 180,E1 -11691.715,E2 -11691.715} C_VEL
LIN {X 0,Y 389.728,Z 347.881,A -85,B 0,C 180,E1 -11693.009,E2 -11693.009} C_VEL
LIN {X 0,Y 389.428,Z 349.678,A -85,B 0,C 180,E1 -11693.784,E2 -11693.784} C_VEL
LIN {X 0,Y 389.439,Z 351.629,A -85,B 0,C 180,E1 -11694.823,E2 -11694.823} C_VEL
LIN {X 0,Y 389.286,Z 353.165,A -85,B 0,C 180,E1 -11695.859,E2 -11695.859} C_VEL
LIN {X 0,Y 389.096,Z 354.306,A -85,B 0,C 180,E1 -11696.894,E2 -11696.894} C_VEL
LIN {X 0,Y 388.952,Z 355.015,A -85,B 0,C 180,E1 -11697.929,E2 -11697.929} C_VEL
LIN {X 0,Y 388.849,Z 355.295,A -85,B 0,C 180,E1 -11698.964,E2 -11698.964} C_VEL
LIN {X 0,Y 388.798,Z 355.181,A -85,B 0,C 180,E1 -11700,E2 -11700} C_VEL
LIN {X 0,Y 388.811,Z 354.662,A -85,B 0,C 180,E1 -11701.036,E2 -11701.036} C_VEL
LIN {X 0,Y 388.89,Z 353.687,A -85,B 0,C 180,E1 -11702.071,E2 -11702.071} C_VEL
LIN {X 0,Y 388.974,Z 352.307,A -85,B 0,C 180,E1 -11703.107,E2 -11703.107} C_VEL
LIN {X 0,Y 388.986,Z 349.424,A -85,B 0,C 180,E1 -11704.664,E2 -11704.664} C_VEL
LIN {X 0,Y 389.196,Z 345.484,A -85,B 0,C 180,E1 -11706.22,E2 -11706.22} C_VEL
LIN {X 0,Y 389.466,Z 340.393,A -85,B 0,C 180,E1 -11707.778,E2 -11707.778} C_VEL
LIN {X 0,Y 389.882,Z 333.991,A -85,B 0,C 180,E1 -11709.337,E2 -11709.337} C_VEL
LIN {X 0,Y 390.411,Z 325.992,A -85,B 0,C 180,E1 -11710.895,E2 -11710.895} C_VEL
LIN {X 0,Y 391.111,Z 316.103,A -85,B 0,C 180,E1 -11712.453,E2 -11712.453} C_VEL
LIN {X 0,Y 391.79,Z 305.849,A -85,B 0,C 180,E1 -11713.75,E2 -11713.75} C_VEL
